KUKA KRL program: ap_0.src, ap_0.dat

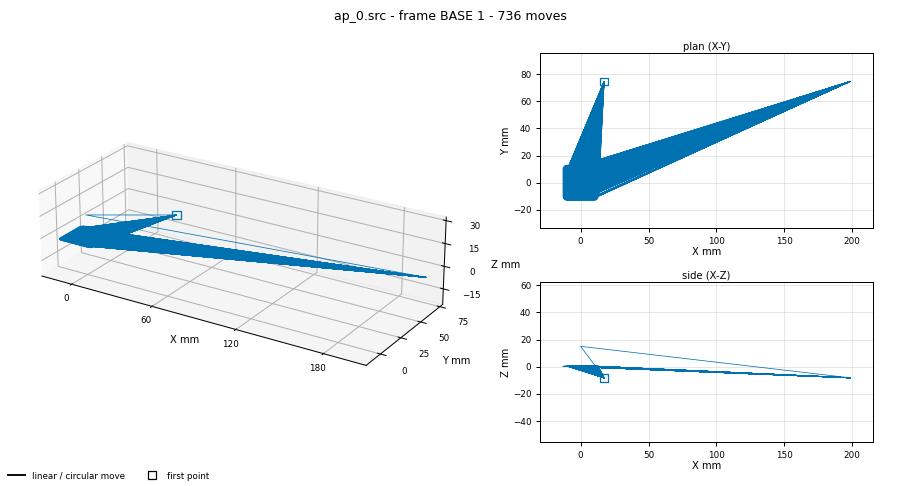
[picture p0: tool path of ap_0.src in frame BASE 1, 736 of 736 moves have a stored position in this frame; points joined in program order, loops and branches not executed]
--- ap_0.src ---
&ACCESS RVP
&REL 65
&PARAM DISKPATH = KRC:\R1\Program
DEF ap_0 ( )
   ;FOLD INI;%{PE}
     ;FOLD BASISTECH INI
       GLOBAL INTERRUPT DECL 3 WHEN $STOPMESS==TRUE DO IR_STOPM ( )
       INTERRUPT ON 3
       BAS (#INITMOV,0 )
     ;ENDFOLD (BASISTECH INI)
     ;FOLD USER INI
       ;Make your modifications here
     ;ENDFOLD (USER INI)
   ;ENDFOLD (INI)

   BAS (#VEL_PTP, 0020.0000)
   BAS (#ACC_PTP, 0020.0000)

   ;-----SET LIN AND ARC MOTION VARIABLES-----
   $VEL.ORI1 = 0350.0000
   $VEL.ORI2 = 0350.0000

   $ACC.CP = 0005.0000
   $ACC.ORI1 = 1000.0000
   $ACC.ORI2 = 1000.0000

   ;-----APPROXIMATION-----
   $APO.CVEL = 0100
   $APO.CPTP = 0100
   $APO.CDIS = 0006.0000
   $APO.CORI = 0090.0000

   BAS (#BASE, 1) ;Positioner
   BAS (#TOOL, 1) ;Vrashatel

   BAS(#VEL_PTP,15)                         ;;Set PTP Axis Velocity
   BAS(#ACC_PTP,50)                         ;;Set PTP Axis Acceleration
   PTP{A1 -92,A2 -133,A3 132,A4 7,A5 50,A6 -10}

;FOLD ARCON WDAT1 LIN P3 Vel=0.5 m/s CPDAT1 Tool[1]:cmttorch Base[1]:vrashatel ;%{PE}
  ;FOLD Parameters ;%{h}
    ;Params IlfProvider=kukaroboter.arctech.arconlin; Kuka.IsGlobalPoint=False; Kuka.PointName=P3; Kuka.BlendingEnabled=False; Kuka.MoveDataName=CPDAT1; Kuka.VelocityPath=0.5; Kuka.CurrentCDSetIndex=0; Kuka.MovementParameterFieldEnabled=True; ArcTech.WdatVarName=WDAT1; ArcTech.Basic=3.4.3.1264
  ;ENDFOLD
  $BWDSTART = FALSE
  LDAT_ACT = LCPDAT1
  FDAT_ACT = FP3
  BAS(#CP_PARAMS, 0.5)
  SET_CD_PARAMS (0)
  TRIGGER WHEN DISTANCE = 1 DELAY = ArcGetDelay(#PreDefinition, WDAT1) DO ArcMainNG(#PreDefinition, WDAT1, WP3) PRIO = -1
  TRIGGER WHEN PATH = ArcGetPath(#OnTheFlyArcOn, WDAT1) DELAY = ArcGetDelay(#GasPreflow, WDAT1) DO ArcMainNG(#GasPreflow, WDAT1, WP3) PRIO = -1
  TRIGGER WHEN PATH = ArcGetPath(#OnTheFlyArcOn, WDAT1) DELAY = 0 DO ArcMainNG(#ArcOnMoveStd, WDAT1, WP3) PRIO = -1
  ArcMainNG(#ArcOnBeforeMoveStd, WDAT1, WP3)
  LIN XP3
  ArcMainNG(#ArcOnAfterMoveStd, WDAT1, WP3)
;ENDFOLD
   $VEL.CP = 0.003
   LIN  {X 0.000, Y 0.000, Z 15.000, A 0.000, B 0.000, C 0.000} C_DIS

;FOLD ARCOFF WDAT2 LIN P4 CPDAT2 Tool[1]:cmttorch Base[1]:vrashatel ;%{PE}
  ;FOLD Parameters ;%{h}
    ;Params IlfProvider=kukaroboter.arctech.arcofflin; Kuka.IsGlobalPoint=False; Kuka.PointName=P4; Kuka.BlendingEnabled=False; Kuka.MoveDataName=CPDAT2; Kuka.VelocityPath=0.01; Kuka.CurrentCDSetIndex=0; Kuka.MovementParameterFieldEnabled=True; ArcTech.WdatVarName=WDAT2; ArcTech.Basic=3.4.3.1264
  ;ENDFOLD
  $BWDSTART = FALSE
  LDAT_ACT = LCPDAT2
  FDAT_ACT = FP4
  BAS(#CP_PARAMS, gArcBasVelDefinition)
  SET_CD_PARAMS (0)
  TRIGGER WHEN PATH = ArcGetPath(#ArcOffBefore, WDAT2) DELAY = 0 DO ArcMainNG(#ArcOffBeforeOffStd, WDAT2, WP4) PRIO = -1
  TRIGGER WHEN PATH = ArcGetPath(#OnTheFlyArcOff, WDAT2) DELAY = 0 DO ArcMainNG(#ArcOffMoveStd, WDAT2, WP4) PRIO = -1
  ArcMainNG(#ArcOffBeforeMoveStd, WDAT2, WP4)
  LIN XP4
  ArcMainNG(#ArcOffAfterMoveStd, WDAT2, WP4)
;ENDFOLD
   $VEL.CP = 0.030
   LIN  {X 13.000, Y -10.000, Z 0.300, A 0.000, B 0.000, C 0.000} C_DIS

;FOLD ARCON WDAT1 LIN P3 Vel=0.5 m/s CPDAT1 Tool[1]:cmttorch Base[1]:vrashatel ;%{PE}
  ;FOLD Parameters ;%{h}
    ;Params IlfProvider=kukaroboter.arctech.arconlin; Kuka.IsGlobalPoint=False; Kuka.PointName=P3; Kuka.BlendingEnabled=False; Kuka.MoveDataName=CPDAT1; Kuka.VelocityPath=0.5; Kuka.CurrentCDSetIndex=0; Kuka.MovementParameterFieldEnabled=True; ArcTech.WdatVarName=WDAT1; ArcTech.Basic=3.4.3.1264
  ;ENDFOLD
  $BWDSTART = FALSE
  LDAT_ACT = LCPDAT1
  FDAT_ACT = FP3
  BAS(#CP_PARAMS, 0.5)
  SET_CD_PARAMS (0)
  TRIGGER WHEN DISTANCE = 1 DELAY = ArcGetDelay(#PreDefinition, WDAT1) DO ArcMainNG(#PreDefinition, WDAT1, WP3) PRIO = -1
  TRIGGER WHEN PATH = ArcGetPath(#OnTheFlyArcOn, WDAT1) DELAY = ArcGetDelay(#GasPreflow, WDAT1) DO ArcMainNG(#GasPreflow, WDAT1, WP3) PRIO = -1
  TRIGGER WHEN PATH = ArcGetPath(#OnTheFlyArcOn, WDAT1) DELAY = 0 DO ArcMainNG(#ArcOnMoveStd, WDAT1, WP3) PRIO = -1
  ArcMainNG(#ArcOnBeforeMoveStd, WDAT1, WP3)
  LIN XP3
  ArcMainNG(#ArcOnAfterMoveStd, WDAT1, WP3)
;ENDFOLD
   $VEL.CP = 0.025
   LIN  {X 13.000, Y -10.000, Z 0.300, A 0.000, B 0.000, C 0.000} C_DIS
   $VEL.CP = 0.030
   LIN  {X 13.000, Y 10.000, Z 0.300, A 0.000, B 0.000, C 0.000} C_DIS
   $VEL.CP = 0.030
   LIN  {X 12.960, Y 10.488, Z 0.300, A 0.000, B 0.000, C 0.000} C_DIS
   $VEL.CP = 0.030
   LIN  {X 12.841, Y 10.963, Z 0.300, A 0.000, B 0.000, C 0.000} C_DIS
   $VEL.CP = 0.030
   LIN  {X 12.647, Y 11.412, Z 0.300, A 0.000, B 0.000, C 0.000} C_DIS
   $VEL.CP = 0.030
   LIN  {X 12.382, Y 11.824, Z 0.300, A 0.000, B 0.000, C 0.000} C_DIS
   $VEL.CP = 0.030
   LIN  {X 12.054, Y 12.187, Z 0.300, A 0.000, B 0.000, C 0.000} C_DIS
   $VEL.CP = 0.030
   LIN  {X 11.671, Y 12.492, Z 0.300, A 0.000, B 0.000, C 0.000} C_DIS
   $VEL.CP = 0.030
   LIN  {X 11.243, Y 12.730, Z 0.300, A 0.000, B 0.000, C 0.000} C_DIS
   $VEL.CP = 0.030
   LIN  {X 10.783, Y 12.896, Z 0.300, A 0.000, B 0.000, C 0.000} C_DIS
   $VEL.CP = 0.030
   LIN  {X 10.302, Y 12.985, Z 0.300, A 0.000, B 0.000, C 0.000} C_DIS
   $VEL.CP = 0.030
   LIN  {X 10.000, Y 13.000, Z 0.300, A 0.000, B 0.000, C 0.000} C_DIS
   $VEL.CP = 0.030
   LIN  {X -10.000, Y 13.000, Z 0.300, A 0.000, B 0.000, C 0.000} C_DIS
   $VEL.CP = 0.030
   LIN  {X -10.488, Y 12.960, Z 0.300, A 0.000, B 0.000, C 0.000} C_DIS
   $VEL.CP = 0.030
   LIN  {X -10.963, Y 12.841, Z 0.300, A 0.000, B 0.000, C 0.000} C_DIS
   $VEL.CP = 0.030
   LIN  {X -11.412, Y 12.647, Z 0.300, A 0.000, B 0.000, C 0.000} C_DIS
   $VEL.CP = 0.030
   LIN  {X -11.824, Y 12.382, Z 0.300, A 0.000, B 0.000, C 0.000} C_DIS
   $VEL.CP = 0.030
   LIN  {X -12.187, Y 12.054, Z 0.300, A 0.000, B 0.000, C 0.000} C_DIS
   $VEL.CP = 0.030
   LIN  {X -12.492, Y 11.671, Z 0.300, A 0.000, B 0.000, C 0.000} C_DIS
   $VEL.CP = 0.030
   LIN  {X -12.730, Y 11.243, Z 0.300, A 0.000, B 0.000, C 0.000} C_DIS
   $VEL.CP = 0.030
   LIN  {X -12.896, Y 10.783, Z 0.300, A 0.000, B 0.000, C 0.000} C_DIS
   $VEL.CP = 0.030
   LIN  {X -12.985, Y 10.302, Z 0.300, A 0.000, B 0.000, C 0.000} C_DIS
   $VEL.CP = 0.030
   LIN  {X -13.000, Y 10.000, Z 0.300, A 0.000, B 0.000, C 0.000} C_DIS
   $VEL.CP = 0.030
   LIN  {X -13.000, Y -10.000, Z 0.300, A 0.000, B 0.000, C 0.000} C_DIS
   $VEL.CP = 0.030
   LIN  {X -12.960, Y -10.488, Z 0.300, A 0.000, B 0.000, C 0.000} C_DIS
   $VEL.CP = 0.030
   LIN  {X -12.841, Y -10.963, Z 0.300, A 0.000, B 0.000, C 0.000} C_DIS
   $VEL.CP = 0.030
   LIN  {X -12.647, Y -11.412, Z 0.300, A 0.000, B 0.000, C 0.000} C_DIS
   $VEL.CP = 0.030
   LIN  {X -12.382, Y -11.824, Z 0.300, A 0.000, B 0.000, C 0.000} C_DIS
   $VEL.CP = 0.030
   LIN  {X -12.054, Y -12.187, Z 0.300, A 0.000, B 0.000, C 0.000} C_DIS
   $VEL.CP = 0.030
   LIN  {X -11.671, Y -12.492, Z 0.300, A 0.000, B 0.000, C 0.000} C_DIS
   $VEL.CP = 0.030
   LIN  {X -11.243, Y -12.730, Z 0.300, A 0.000, B 0.000, C 0.000} C_DIS
   $VEL.CP = 0.030
   LIN  {X -10.783, Y -12.896, Z 0.300, A 0.000, B 0.000, C 0.000} C_DIS
   $VEL.CP = 0.030
   LIN  {X -10.302, Y -12.985, Z 0.300, A 0.000, B 0.000, C 0.000} C_DIS
   $VEL.CP = 0.030
   LIN  {X -10.000, Y -13.000, Z 0.300, A 0.000, B 0.000, C 0.000} C_DIS
   $VEL.CP = 0.030
   LIN  {X 10.000, Y -13.000, Z 0.300, A 0.000, B 0.000, C 0.000} C_DIS
   $VEL.CP = 0.030
   LIN  {X 10.488, Y -12.960, Z 0.300, A 0.000, B 0.000, C 0.000} C_DIS
   $VEL.CP = 0.030
   LIN  {X 10.963, Y -12.841, Z 0.300, A 0.000, B 0.000, C 0.000} C_DIS
   $VEL.CP = 0.030
   LIN  {X 11.412, Y -12.647, Z 0.300, A 0.000, B 0.000, C 0.000} C_DIS
   $VEL.CP = 0.030
   LIN  {X 11.824, Y -12.382, Z 0.300, A 0.000, B 0.000, C 0.000} C_DIS
   $VEL.CP = 0.030
   LIN  {X 12.187, Y -12.054, Z 0.300, A 0.000, B 0.000, C 0.000} C_DIS
   $VEL.CP = 0.030
   LIN  {X 12.492, Y -11.671, Z 0.300, A 0.000, B 0.000, C 0.000} C_DIS
   $VEL.CP = 0.030
   LIN  {X 12.730, Y -11.243, Z 0.300, A 0.000, B 0.000, C 0.000} C_DIS
   $VEL.CP = 0.030
   LIN  {X 12.896, Y -10.783, Z 0.300, A 0.000, B 0.000, C 0.000} C_DIS
   $VEL.CP = 0.030
   LIN  {X 12.985, Y -10.302, Z 0.300, A 0.000, B 0.000, C 0.000} C_DIS
   $VEL.CP = 0.030
   LIN  {X 13.000, Y -10.000, Z 0.300, A 0.000, B 0.000, C 0.000} C_DIS

;FOLD ARCOFF WDAT2 LIN P4 CPDAT2 Tool[1]:cmttorch Base[1]:vrashatel ;%{PE}
  ;FOLD Parameters ;%{h}
    ;Params IlfProvider=kukaroboter.arctech.arcofflin; Kuka.IsGlobalPoint=False; Kuka.PointName=P4; Kuka.BlendingEnabled=False; Kuka.MoveDataName=CPDAT2; Kuka.VelocityPath=0.01; Kuka.CurrentCDSetIndex=0; Kuka.MovementParameterFieldEnabled=True; ArcTech.WdatVarName=WDAT2; ArcTech.Basic=3.4.3.1264
  ;ENDFOLD
  $BWDSTART = FALSE
  LDAT_ACT = LCPDAT2
  FDAT_ACT = FP4
  BAS(#CP_PARAMS, gArcBasVelDefinition)
  SET_CD_PARAMS (0)
  TRIGGER WHEN PATH = ArcGetPath(#ArcOffBefore, WDAT2) DELAY = 0 DO ArcMainNG(#ArcOffBeforeOffStd, WDAT2, WP4) PRIO = -1
  TRIGGER WHEN PATH = ArcGetPath(#OnTheFlyArcOff, WDAT2) DELAY = 0 DO ArcMainNG(#ArcOffMoveStd, WDAT2, WP4) PRIO = -1
  ArcMainNG(#ArcOffBeforeMoveStd, WDAT2, WP4)
  LIN XP4
  ArcMainNG(#ArcOffAfterMoveStd, WDAT2, WP4)
;ENDFOLD
   $VEL.CP = 0.030
   LIN  {X 12.600, Y -10.000, Z 0.300, A 0.000, B 0.000, C 0.000} C_DIS

;FOLD ARCON WDAT1 LIN P3 Vel=0.5 m/s CPDAT1 Tool[1]:cmttorch Base[1]:vrashatel ;%{PE}
  ;FOLD Parameters ;%{h}
    ;Params IlfProvider=kukaroboter.arctech.arconlin; Kuka.IsGlobalPoint=False; Kuka.PointName=P3; Kuka.BlendingEnabled=False; Kuka.MoveDataName=CPDAT1; Kuka.VelocityPath=0.5; Kuka.CurrentCDSetIndex=0; Kuka.MovementParameterFieldEnabled=True; ArcTech.WdatVarName=WDAT1; ArcTech.Basic=3.4.3.1264
  ;ENDFOLD
  $BWDSTART = FALSE
  LDAT_ACT = LCPDAT1
  FDAT_ACT = FP3
  BAS(#CP_PARAMS, 0.5)
  SET_CD_PARAMS (0)
  TRIGGER WHEN DISTANCE = 1 DELAY = ArcGetDelay(#PreDefinition, WDAT1) DO ArcMainNG(#PreDefinition, WDAT1, WP3) PRIO = -1
  TRIGGER WHEN PATH = ArcGetPath(#OnTheFlyArcOn, WDAT1) DELAY = ArcGetDelay(#GasPreflow, WDAT1) DO ArcMainNG(#GasPreflow, WDAT1, WP3) PRIO = -1
  TRIGGER WHEN PATH = ArcGetPath(#OnTheFlyArcOn, WDAT1) DELAY = 0 DO ArcMainNG(#ArcOnMoveStd, WDAT1, WP3) PRIO = -1
  ArcMainNG(#ArcOnBeforeMoveStd, WDAT1, WP3)
  LIN XP3
  ArcMainNG(#ArcOnAfterMoveStd, WDAT1, WP3)
;ENDFOLD
   $VEL.CP = 0.030
   LIN  {X 12.600, Y 10.000, Z 0.300, A 0.000, B 0.000, C 0.000} C_DIS
   $VEL.CP = 0.030
   LIN  {X 12.560, Y 10.454, Z 0.300, A 0.000, B 0.000, C 0.000} C_DIS
   $VEL.CP = 0.030
   LIN  {X 12.442, Y 10.894, Z 0.300, A 0.000, B 0.000, C 0.000} C_DIS
   $VEL.CP = 0.030
   LIN  {X 12.248, Y 11.306, Z 0.300, A 0.000, B 0.000, C 0.000} C_DIS
   $VEL.CP = 0.030
   LIN  {X 11.985, Y 11.679, Z 0.300, A 0.000, B 0.000, C 0.000} C_DIS
   $VEL.CP = 0.030
   LIN  {X 11.662, Y 12.000, Z 0.300, A 0.000, B 0.000, C 0.000} C_DIS
   $VEL.CP = 0.030
   LIN  {X 11.287, Y 12.259, Z 0.300, A 0.000, B 0.000, C 0.000} C_DIS
   $VEL.CP = 0.030
   LIN  {X 10.873, Y 12.449, Z 0.300, A 0.000, B 0.000, C 0.000} C_DIS
   $VEL.CP = 0.030
   LIN  {X 10.432, Y 12.564, Z 0.300, A 0.000, B 0.000, C 0.000} C_DIS
   $VEL.CP = 0.030
   LIN  {X 10.000, Y 12.600, Z 0.300, A 0.000, B 0.000, C 0.000} C_DIS
   $VEL.CP = 0.030
   LIN  {X -10.000, Y 12.600, Z 0.300, A 0.000, B 0.000, C 0.000} C_DIS
   $VEL.CP = 0.030
   LIN  {X -10.454, Y 12.560, Z 0.300, A 0.000, B 0.000, C 0.000} C_DIS
   $VEL.CP = 0.030
   LIN  {X -10.894, Y 12.442, Z 0.300, A 0.000, B 0.000, C 0.000} C_DIS
   $VEL.CP = 0.030
   LIN  {X -11.306, Y 12.248, Z 0.300, A 0.000, B 0.000, C 0.000} C_DIS
   $VEL.CP = 0.030
   LIN  {X -11.679, Y 11.985, Z 0.300, A 0.000, B 0.000, C 0.000} C_DIS
   $VEL.CP = 0.030
   LIN  {X -12.000, Y 11.662, Z 0.300, A 0.000, B 0.000, C 0.000} C_DIS
   $VEL.CP = 0.030
   LIN  {X -12.259, Y 11.287, Z 0.300, A 0.000, B 0.000, C 0.000} C_DIS
   $VEL.CP = 0.030
   LIN  {X -12.449, Y 10.873, Z 0.300, A 0.000, B 0.000, C 0.000} C_DIS
   $VEL.CP = 0.030
   LIN  {X -12.564, Y 10.432, Z 0.300, A 0.000, B 0.000, C 0.000} C_DIS
   $VEL.CP = 0.030
   LIN  {X -12.600, Y 10.000, Z 0.300, A 0.000, B 0.000, C 0.000} C_DIS
   $VEL.CP = 0.030
   LIN  {X -12.600, Y -10.000, Z 0.300, A 0.000, B 0.000, C 0.000} C_DIS
   $VEL.CP = 0.030
   LIN  {X -12.560, Y -10.454, Z 0.300, A 0.000, B 0.000, C 0.000} C_DIS
   $VEL.CP = 0.030
   LIN  {X -12.442, Y -10.894, Z 0.300, A 0.000, B 0.000, C 0.000} C_DIS
   $VEL.CP = 0.030
   LIN  {X -12.248, Y -11.306, Z 0.300, A 0.000, B 0.000, C 0.000} C_DIS
   $VEL.CP = 0.030
   LIN  {X -11.985, Y -11.679, Z 0.300, A 0.000, B 0.000, C 0.000} C_DIS
   $VEL.CP = 0.030
   LIN  {X -11.662, Y -12.000, Z 0.300, A 0.000, B 0.000, C 0.000} C_DIS
   $VEL.CP = 0.030
   LIN  {X -11.287, Y -12.259, Z 0.300, A 0.000, B 0.000, C 0.000} C_DIS
   $VEL.CP = 0.030
   LIN  {X -10.873, Y -12.449, Z 0.300, A 0.000, B 0.000, C 0.000} C_DIS
   $VEL.CP = 0.030
   LIN  {X -10.432, Y -12.564, Z 0.300, A 0.000, B 0.000, C 0.000} C_DIS
   $VEL.CP = 0.030
   LIN  {X -10.000, Y -12.600, Z 0.300, A 0.000, B 0.000, C 0.000} C_DIS
   $VEL.CP = 0.030
   LIN  {X 10.000, Y -12.600, Z 0.300, A 0.000, B 0.000, C 0.000} C_DIS
   $VEL.CP = 0.030
   LIN  {X 10.454, Y -12.560, Z 0.300, A 0.000, B 0.000, C 0.000} C_DIS
   $VEL.CP = 0.030
   LIN  {X 10.894, Y -12.442, Z 0.300, A 0.000, B 0.000, C 0.000} C_DIS
   $VEL.CP = 0.030
   LIN  {X 11.306, Y -12.248, Z 0.300, A 0.000, B 0.000, C 0.000} C_DIS
   $VEL.CP = 0.030
   LIN  {X 11.679, Y -11.985, Z 0.300, A 0.000, B 0.000, C 0.000} C_DIS
   $VEL.CP = 0.030
   LIN  {X 12.000, Y -11.662, Z 0.300, A 0.000, B 0.000, C 0.000} C_DIS
   $VEL.CP = 0.030
   LIN  {X 12.259, Y -11.287, Z 0.300, A 0.000, B 0.000, C 0.000} C_DIS
   $VEL.CP = 0.030
   LIN  {X 12.449, Y -10.873, Z 0.300, A 0.000, B 0.000, C 0.000} C_DIS
   $VEL.CP = 0.030
   LIN  {X 12.564, Y -10.432, Z 0.300, A 0.000, B 0.000, C 0.000} C_DIS
   $VEL.CP = 0.030
   LIN  {X 12.600, Y -10.000, Z 0.300, A 0.000, B 0.000, C 0.000} C_DIS

;FOLD ARCOFF WDAT2 LIN P4 CPDAT2 Tool[1]:cmttorch Base[1]:vrashatel ;%{PE}
  ;FOLD Parameters ;%{h}
    ;Params IlfProvider=kukaroboter.arctech.arcofflin; Kuka.IsGlobalPoint=False; Kuka.PointName=P4; Kuka.BlendingEnabled=False; Kuka.MoveDataName=CPDAT2; Kuka.VelocityPath=0.01; Kuka.CurrentCDSetIndex=0; Kuka.MovementParameterFieldEnabled=True; ArcTech.WdatVarName=WDAT2; ArcTech.Basic=3.4.3.1264
  ;ENDFOLD
  $BWDSTART = FALSE
  LDAT_ACT = LCPDAT2
  FDAT_ACT = FP4
  BAS(#CP_PARAMS, gArcBasVelDefinition)
  SET_CD_PARAMS (0)
  TRIGGER WHEN PATH = ArcGetPath(#ArcOffBefore, WDAT2) DELAY = 0 DO ArcMainNG(#ArcOffBeforeOffStd, WDAT2, WP4) PRIO = -1
  TRIGGER WHEN PATH = ArcGetPath(#OnTheFlyArcOff, WDAT2) DELAY = 0 DO ArcMainNG(#ArcOffMoveStd, WDAT2, WP4) PRIO = -1
  ArcMainNG(#ArcOffBeforeMoveStd, WDAT2, WP4)
  LIN XP4
  ArcMainNG(#ArcOffAfterMoveStd, WDAT2, WP4)
;ENDFOLD
   $VEL.CP = 0.030
   LIN  {X 12.200, Y -10.000, Z 0.300, A 0.000, B 0.000, C 0.000} C_DIS

;FOLD ARCON WDAT1 LIN P3 Vel=0.5 m/s CPDAT1 Tool[1]:cmttorch Base[1]:vrashatel ;%{PE}
  ;FOLD Parameters ;%{h}
    ;Params IlfProvider=kukaroboter.arctech.arconlin; Kuka.IsGlobalPoint=False; Kuka.PointName=P3; Kuka.BlendingEnabled=False; Kuka.MoveDataName=CPDAT1; Kuka.VelocityPath=0.5; Kuka.CurrentCDSetIndex=0; Kuka.MovementParameterFieldEnabled=True; ArcTech.WdatVarName=WDAT1; ArcTech.Basic=3.4.3.1264
  ;ENDFOLD
  $BWDSTART = FALSE
  LDAT_ACT = LCPDAT1
  FDAT_ACT = FP3
  BAS(#CP_PARAMS, 0.5)
  SET_CD_PARAMS (0)
  TRIGGER WHEN DISTANCE = 1 DELAY = ArcGetDelay(#PreDefinition, WDAT1) DO ArcMainNG(#PreDefinition, WDAT1, WP3) PRIO = -1
  TRIGGER WHEN PATH = ArcGetPath(#OnTheFlyArcOn, WDAT1) DELAY = ArcGetDelay(#GasPreflow, WDAT1) DO ArcMainNG(#GasPreflow, WDAT1, WP3) PRIO = -1
  TRIGGER WHEN PATH = ArcGetPath(#OnTheFlyArcOn, WDAT1) DELAY = 0 DO ArcMainNG(#ArcOnMoveStd, WDAT1, WP3) PRIO = -1
  ArcMainNG(#ArcOnBeforeMoveStd, WDAT1, WP3)
  LIN XP3
  ArcMainNG(#ArcOnAfterMoveStd, WDAT1, WP3)
;ENDFOLD
   $VEL.CP = 0.030
   LIN  {X 12.200, Y 10.000, Z 0.300, A 0.000, B 0.000, C 0.000} C_DIS
   $VEL.CP = 0.030
   LIN  {X 12.160, Y 10.417, Z 0.300, A 0.000, B 0.000, C 0.000} C_DIS
   $VEL.CP = 0.030
   LIN  {X 12.042, Y 10.819, Z 0.300, A 0.000, B 0.000, C 0.000} C_DIS
   $VEL.CP = 0.030
   LIN  {X 11.849, Y 11.191, Z 0.300, A 0.000, B 0.000, C 0.000} C_DIS
   $VEL.CP = 0.030
   LIN  {X 11.590, Y 11.520, Z 0.300, A 0.000, B 0.000, C 0.000} C_DIS
   $VEL.CP = 0.030
   LIN  {X 11.273, Y 11.794, Z 0.300, A 0.000, B 0.000, C 0.000} C_DIS
   $VEL.CP = 0.030
   LIN  {X 10.910, Y 12.003, Z 0.300, A 0.000, B 0.000, C 0.000} C_DIS
   $VEL.CP = 0.030
   LIN  {X 10.513, Y 12.139, Z 0.300, A 0.000, B 0.000, C 0.000} C_DIS
   $VEL.CP = 0.030
   LIN  {X 10.000, Y 12.200, Z 0.300, A 0.000, B 0.000, C 0.000} C_DIS
   $VEL.CP = 0.030
   LIN  {X -10.000, Y 12.200, Z 0.300, A 0.000, B 0.000, C 0.000} C_DIS
   $VEL.CP = 0.030
   LIN  {X -10.417, Y 12.160, Z 0.300, A 0.000, B 0.000, C 0.000} C_DIS
   $VEL.CP = 0.030
   LIN  {X -10.819, Y 12.042, Z 0.300, A 0.000, B 0.000, C 0.000} C_DIS
   $VEL.CP = 0.030
   LIN  {X -11.191, Y 11.849, Z 0.300, A 0.000, B 0.000, C 0.000} C_DIS
   $VEL.CP = 0.030
   LIN  {X -11.520, Y 11.590, Z 0.300, A 0.000, B 0.000, C 0.000} C_DIS
   $VEL.CP = 0.030
   LIN  {X -11.794, Y 11.273, Z 0.300, A 0.000, B 0.000, C 0.000} C_DIS
   $VEL.CP = 0.030
   LIN  {X -12.003, Y 10.910, Z 0.300, A 0.000, B 0.000, C 0.000} C_DIS
   $VEL.CP = 0.030
   LIN  {X -12.139, Y 10.513, Z 0.300, A 0.000, B 0.000, C 0.000} C_DIS
   $VEL.CP = 0.030
   LIN  {X -12.200, Y 10.000, Z 0.300, A 0.000, B 0.000, C 0.000} C_DIS
   $VEL.CP = 0.030
   LIN  {X -12.200, Y -10.000, Z 0.300, A 0.000, B 0.000, C 0.000} C_DIS
   $VEL.CP = 0.030
   LIN  {X -12.160, Y -10.417, Z 0.300, A 0.000, B 0.000, C 0.000} C_DIS
   $VEL.CP = 0.030
   LIN  {X -12.042, Y -10.819, Z 0.300, A 0.000, B 0.000, C 0.000} C_DIS
   $VEL.CP = 0.030
   LIN  {X -11.849, Y -11.191, Z 0.300, A 0.000, B 0.000, C 0.000} C_DIS
   $VEL.CP = 0.030
   LIN  {X -11.590, Y -11.520, Z 0.300, A 0.000, B 0.000, C 0.000} C_DIS
   $VEL.CP = 0.030
   LIN  {X -11.273, Y -11.794, Z 0.300, A 0.000, B 0.000, C 0.000} C_DIS
   $VEL.CP = 0.030
   LIN  {X -10.910, Y -12.003, Z 0.300, A 0.000, B 0.000, C 0.000} C_DIS
   $VEL.CP = 0.030
   LIN  {X -10.513, Y -12.139, Z 0.300, A 0.000, B 0.000, C 0.000} C_DIS
   $VEL.CP = 0.030
   LIN  {X -10.000, Y -12.200, Z 0.300, A 0.000, B 0.000, C 0.000} C_DIS
   $VEL.CP = 0.030
   LIN  {X 10.000, Y -12.200, Z 0.300, A 0.000, B 0.000, C 0.000} C_DIS
   $VEL.CP = 0.030
   LIN  {X 10.417, Y -12.160, Z 0.300, A 0.000, B 0.000, C 0.000} C_DIS
   $VEL.CP = 0.030
   LIN  {X 10.819, Y -12.042, Z 0.300, A 0.000, B 0.000, C 0.000} C_DIS
   $VEL.CP = 0.030
   LIN  {X 11.191, Y -11.849, Z 0.300, A 0.000, B 0.000, C 0.000} C_DIS
   $VEL.CP = 0.030
   LIN  {X 11.520, Y -11.590, Z 0.300, A 0.000, B 0.000, C 0.000} C_DIS
   $VEL.CP = 0.030
   LIN  {X 11.794, Y -11.273, Z 0.300, A 0.000, B 0.000, C 0.000} C_DIS
   $VEL.CP = 0.030
   LIN  {X 12.003, Y -10.910, Z 0.300, A 0.000, B 0.000, C 0.000} C_DIS
   $VEL.CP = 0.030
   LIN  {X 12.139, Y -10.513, Z 0.300, A 0.000, B 0.000, C 0.000} C_DIS
   $VEL.CP = 0.030
   LIN  {X 12.200, Y -10.000, Z 0.300, A 0.000, B 0.000, C 0.000} C_DIS

;FOLD ARCOFF WDAT2 LIN P4 CPDAT2 Tool[1]:cmttorch Base[1]:vrashatel ;%{PE}
  ;FOLD Parameters ;%{h}
    ;Params IlfProvider=kukaroboter.arctech.arcofflin; Kuka.IsGlobalPoint=False; Kuka.PointName=P4; Kuka.BlendingEnabled=False; Kuka.MoveDataName=CPDAT2; Kuka.VelocityPath=0.01; Kuka.CurrentCDSetIndex=0; Kuka.MovementParameterFieldEnabled=True; ArcTech.WdatVarName=WDAT2; ArcTech.Basic=3.4.3.1264
  ;ENDFOLD
  $BWDSTART = FALSE
  LDAT_ACT = LCPDAT2
  FDAT_ACT = FP4
  BAS(#CP_PARAMS, gArcBasVelDefinition)
  SET_CD_PARAMS (0)
  TRIGGER WHEN PATH = ArcGetPath(#ArcOffBefore, WDAT2) DELAY = 0 DO ArcMainNG(#ArcOffBeforeOffStd, WDAT2, WP4) PRIO = -1
  TRIGGER WHEN PATH = ArcGetPath(#OnTheFlyArcOff, WDAT2) DELAY = 0 DO ArcMainNG(#ArcOffMoveStd, WDAT2, WP4) PRIO = -1
  ArcMainNG(#ArcOffBeforeMoveStd, WDAT2, WP4)
  LIN XP4
  ArcMainNG(#ArcOffAfterMoveStd, WDAT2, WP4)
;ENDFOLD
   $VEL.CP = 0.030
   LIN  {X 11.800, Y -10.000, Z 0.300, A 0.000, B 0.000, C 0.000} C_DIS

;FOLD ARCON WDAT1 LIN P3 Vel=0.5 m/s CPDAT1 Tool[1]:cmttorch Base[1]:vrashatel ;%{PE}
  ;FOLD Parameters ;%{h}
    ;Params IlfProvider=kukaroboter.arctech.arconlin; Kuka.IsGlobalPoint=False; Kuka.PointName=P3; Kuka.BlendingEnabled=False; Kuka.MoveDataName=CPDAT1; Kuka.VelocityPath=0.5; Kuka.CurrentCDSetIndex=0; Kuka.MovementParameterFieldEnabled=True; ArcTech.WdatVarName=WDAT1; ArcTech.Basic=3.4.3.1264
  ;ENDFOLD
  $BWDSTART = FALSE
  LDAT_ACT = LCPDAT1
  FDAT_ACT = FP3
  BAS(#CP_PARAMS, 0.5)
  SET_CD_PARAMS (0)
  TRIGGER WHEN DISTANCE = 1 DELAY = ArcGetDelay(#PreDefinition, WDAT1) DO ArcMainNG(#PreDefinition, WDAT1, WP3) PRIO = -1
  TRIGGER WHEN PATH = ArcGetPath(#OnTheFlyArcOn, WDAT1) DELAY = ArcGetDelay(#GasPreflow, WDAT1) DO ArcMainNG(#GasPreflow, WDAT1, WP3) PRIO = -1
  TRIGGER WHEN PATH = ArcGetPath(#OnTheFlyArcOn, WDAT1) DELAY = 0 DO ArcMainNG(#ArcOnMoveStd, WDAT1, WP3) PRIO = -1
  ArcMainNG(#ArcOnBeforeMoveStd, WDAT1, WP3)
  LIN XP3
  ArcMainNG(#ArcOnAfterMoveStd, WDAT1, WP3)
;ENDFOLD
   $VEL.CP = 0.030
   LIN  {X 11.800, Y 10.000, Z 0.300, A 0.000, B 0.000, C 0.000} C_DIS
   $VEL.CP = 0.030
   LIN  {X 11.760, Y 10.377, Z 0.300, A 0.000, B 0.000, C 0.000} C_DIS
   $VEL.CP = 0.030
   LIN  {X 11.642, Y 10.737, Z 0.300, A 0.000, B 0.000, C 0.000} C_DIS
   $VEL.CP = 0.030
   LIN  {X 11.452, Y 11.064, Z 0.300, A 0.000, B 0.000, C 0.000} C_DIS
   $VEL.CP = 0.030
   LIN  {X 11.197, Y 11.345, Z 0.300, A 0.000, B 0.000, C 0.000} C_DIS
   $VEL.CP = 0.030
   LIN  {X 10.888, Y 11.565, Z 0.300, A 0.000, B 0.000, C 0.000} C_DIS
   $VEL.CP = 0.030
   LIN  {X 10.541, Y 11.717, Z 0.300, A 0.000, B 0.000, C 0.000} C_DIS
   $VEL.CP = 0.030
   LIN  {X 10.000, Y 11.800, Z 0.300, A 0.000, B 0.000, C 0.000} C_DIS
   $VEL.CP = 0.030
   LIN  {X -10.000, Y 11.800, Z 0.300, A 0.000, B 0.000, C 0.000} C_DIS
   $VEL.CP = 0.030
   LIN  {X -10.377, Y 11.760, Z 0.300, A 0.000, B 0.000, C 0.000} C_DIS
   $VEL.CP = 0.030
   LIN  {X -10.737, Y 11.642, Z 0.300, A 0.000, B 0.000, C 0.000} C_DIS
   $VEL.CP = 0.030
   LIN  {X -11.064, Y 11.452, Z 0.300, A 0.000, B 0.000, C 0.000} C_DIS
   $VEL.CP = 0.030
   LIN  {X -11.345, Y 11.197, Z 0.300, A 0.000, B 0.000, C 0.000} C_DIS
   $VEL.CP = 0.030
   LIN  {X -11.565, Y 10.888, Z 0.300, A 0.000, B 0.000, C 0.000} C_DIS
   $VEL.CP = 0.030
   LIN  {X -11.717, Y 10.541, Z 0.300, A 0.000, B 0.000, C 0.000} C_DIS
   $VEL.CP = 0.030
   LIN  {X -11.800, Y 10.000, Z 0.300, A 0.000, B 0.000, C 0.000} C_DIS
   $VEL.CP = 0.030
   LIN  {X -11.800, Y -10.000, Z 0.300, A 0.000, B 0.000, C 0.000} C_DIS
   $VEL.CP = 0.030
   LIN  {X -11.760, Y -10.377, Z 0.300, A 0.000, B 0.000, C 0.000} C_DIS
   $VEL.CP = 0.030
   LIN  {X -11.642, Y -10.737, Z 0.300, A 0.000, B 0.000, C 0.000} C_DIS
   $VEL.CP = 0.030
   LIN  {X -11.452, Y -11.064, Z 0.300, A 0.000, B 0.000, C 0.000} C_DIS
   $VEL.CP = 0.030
   LIN  {X -11.197, Y -11.345, Z 0.300, A 0.000, B 0.000, C 0.000} C_DIS
   $VEL.CP = 0.030
   LIN  {X -10.888, Y -11.565, Z 0.300, A 0.000, B 0.000, C 0.000} C_DIS
   $VEL.CP = 0.030
   LIN  {X -10.541, Y -11.717, Z 0.300, A 0.000, B 0.000, C 0.000} C_DIS
   $VEL.CP = 0.030
   LIN  {X -10.000, Y -11.800, Z 0.300, A 0.000, B 0.000, C 0.000} C_DIS
   $VEL.CP = 0.030
   LIN  {X 10.000, Y -11.800, Z 0.300, A 0.000, B 0.000, C 0.000} C_DIS
   $VEL.CP = 0.030
   LIN  {X 10.377, Y -11.760, Z 0.300, A 0.000, B 0.000, C 0.000} C_DIS
   $VEL.CP = 0.030
   LIN  {X 10.737, Y -11.642, Z 0.300, A 0.000, B 0.000, C 0.000} C_DIS
   $VEL.CP = 0.030
   LIN  {X 11.064, Y -11.452, Z 0.300, A 0.000, B 0.000, C 0.000} C_DIS
   $VEL.CP = 0.030
   LIN  {X 11.345, Y -11.197, Z 0.300, A 0.000, B 0.000, C 0.000} C_DIS
   $VEL.CP = 0.030
   LIN  {X 11.565, Y -10.888, Z 0.300, A 0.000, B 0.000, C 0.000} C_DIS
   $VEL.CP = 0.030
   LIN  {X 11.717, Y -10.541, Z 0.300, A 0.000, B 0.000, C 0.000} C_DIS
   $VEL.CP = 0.030
   LIN  {X 11.800, Y -10.000, Z 0.300, A 0.000, B 0.000, C 0.000} C_DIS

;FOLD ARCOFF WDAT2 LIN P4 CPDAT2 Tool[1]:cmttorch Base[1]:vrashatel ;%{PE}
  ;FOLD Parameters ;%{h}
    ;Params IlfProvider=kukaroboter.arctech.arcofflin; Kuka.IsGlobalPoint=False; Kuka.PointName=P4; Kuka.BlendingEnabled=False; Kuka.MoveDataName=CPDAT2; Kuka.VelocityPath=0.01; Kuka.CurrentCDSetIndex=0; Kuka.MovementParameterFieldEnabled=True; ArcTech.WdatVarName=WDAT2; ArcTech.Basic=3.4.3.1264
  ;ENDFOLD
  $BWDSTART = FALSE
  LDAT_ACT = LCPDAT2
  FDAT_ACT = FP4
  BAS(#CP_PARAMS, gArcBasVelDefinition)
  SET_CD_PARAMS (0)
  TRIGGER WHEN PATH = ArcGetPath(#ArcOffBefore, WDAT2) DELAY = 0 DO ArcMainNG(#ArcOffBeforeOffStd, WDAT2, WP4) PRIO = -1
  TRIGGER WHEN PATH = ArcGetPath(#OnTheFlyArcOff, WDAT2) DELAY = 0 DO ArcMainNG(#ArcOffMoveStd, WDAT2, WP4) PRIO = -1
  ArcMainNG(#ArcOffBeforeMoveStd, WDAT2, WP4)
  LIN XP4
  ArcMainNG(#ArcOffAfterMoveStd, WDAT2, WP4)
;ENDFOLD
   $VEL.CP = 0.030
   LIN  {X 11.400, Y -10.000, Z 0.300, A 0.000, B 0.000, C 0.000} C_DIS

;FOLD ARCON WDAT1 LIN P3 Vel=0.5 m/s CPDAT1 Tool[1]:cmttorch Base[1]:vrashatel ;%{PE}
  ;FOLD Parameters ;%{h}
    ;Params IlfProvider=kukaroboter.arctech.arconlin; Kuka.IsGlobalPoint=False; Kuka.PointName=P3; Kuka.BlendingEnabled=False; Kuka.MoveDataName=CPDAT1; Kuka.VelocityPath=0.5; Kuka.CurrentCDSetIndex=0; Kuka.MovementParameterFieldEnabled=True; ArcTech.WdatVarName=WDAT1; ArcTech.Basic=3.4.3.1264
  ;ENDFOLD
  $BWDSTART = FALSE
  LDAT_ACT = LCPDAT1
  FDAT_ACT = FP3
  BAS(#CP_PARAMS, 0.5)
  SET_CD_PARAMS (0)
  TRIGGER WHEN DISTANCE = 1 DELAY = ArcGetDelay(#PreDefinition, WDAT1) DO ArcMainNG(#PreDefinition, WDAT1, WP3) PRIO = -1
  TRIGGER WHEN PATH = ArcGetPath(#OnTheFlyArcOn, WDAT1) DELAY = ArcGetDelay(#GasPreflow, WDAT1) DO ArcMainNG(#GasPreflow, WDAT1, WP3) PRIO = -1
  TRIGGER WHEN PATH = ArcGetPath(#OnTheFlyArcOn, WDAT1) DELAY = 0 DO ArcMainNG(#ArcOnMoveStd, WDAT1, WP3) PRIO = -1
  ArcMainNG(#ArcOnBeforeMoveStd, WDAT1, WP3)
  LIN XP3
  ArcMainNG(#ArcOnAfterMoveStd, WDAT1, WP3)
;ENDFOLD
   $VEL.CP = 0.030
   LIN  {X 11.400, Y 10.000, Z 0.300, A 0.000, B 0.000, C 0.000} C_DIS
   $VEL.CP = 0.030
   LIN  {X 11.360, Y 10.332, Z 0.300, A 0.000, B 0.000, C 0.000} C_DIS
   $VEL.CP = 0.030
   LIN  {X 11.243, Y 10.644, Z 0.300, A 0.000, B 0.000, C 0.000} C_DIS
   $VEL.CP = 0.030
   LIN  {X 11.055, Y 10.921, Z 0.300, A 0.000, B 0.000, C 0.000} C_DIS
   $VEL.CP = 0.030
   LIN  {X 10.807, Y 11.144, Z 0.300, A 0.000, B 0.000, C 0.000} C_DIS
   $VEL.CP = 0.030
   LIN  {X 10.513, Y 11.303, Z 0.300, A 0.000, B 0.000, C 0.000} C_DIS
   $VEL.CP = 0.030
   LIN  {X 10.189, Y 11.387, Z 0.300, A 0.000, B 0.000, C 0.000} C_DIS
   $VEL.CP = 0.030
   LIN  {X 10.000, Y 11.400, Z 0.300, A 0.000, B 0.000, C 0.000} C_DIS
   $VEL.CP = 0.030
   LIN  {X -10.000, Y 11.400, Z 0.300, A 0.000, B 0.000, C 0.000} C_DIS
   $VEL.CP = 0.030
   LIN  {X -10.332, Y 11.360, Z 0.300, A 0.000, B 0.000, C 0.000} C_DIS
   $VEL.CP = 0.030
   LIN  {X -10.644, Y 11.243, Z 0.300, A 0.000, B 0.000, C 0.000} C_DIS
   $VEL.CP = 0.030
   LIN  {X -10.921, Y 11.055, Z 0.300, A 0.000, B 0.000, C 0.000} C_DIS
   $VEL.CP = 0.030
   LIN  {X -11.144, Y 10.807, Z 0.300, A 0.000, B 0.000, C 0.000} C_DIS
   $VEL.CP = 0.030
   LIN  {X -11.303, Y 10.513, Z 0.300, A 0.000, B 0.000, C 0.000} C_DIS
   $VEL.CP = 0.030
   LIN  {X -11.387, Y 10.189, Z 0.300, A 0.000, B 0.000, C 0.000} C_DIS
   $VEL.CP = 0.030
   LIN  {X -11.400, Y 10.000, Z 0.300, A 0.000, B 0.000, C 0.000} C_DIS
   $VEL.CP = 0.030
   LIN  {X -11.400, Y -10.000, Z 0.300, A 0.000, B 0.000, C 0.000} C_DIS
   $VEL.CP = 0.030
   LIN  {X -11.360, Y -10.332, Z 0.300, A 0.000, B 0.000, C 0.000} C_DIS
   $VEL.CP = 0.030
   LIN  {X -11.243, Y -10.644, Z 0.300, A 0.000, B 0.000, C 0.000} C_DIS
   $VEL.CP = 0.030
   LIN  {X -11.055, Y -10.921, Z 0.300, A 0.000, B 0.000, C 0.000} C_DIS
   $VEL.CP = 0.030
   LIN  {X -10.807, Y -11.144, Z 0.300, A 0.000, B 0.000, C 0.000} C_DIS
   $VEL.CP = 0.030
   LIN  {X -10.513, Y -11.303, Z 0.300, A 0.000, B 0.000, C 0.000} C_DIS
   $VEL.CP = 0.030
   LIN  {X -10.189, Y -11.387, Z 0.300, A 0.000, B 0.000, C 0.000} C_DIS
   $VEL.CP = 0.030
   LIN  {X -10.000, Y -11.400, Z 0.300, A 0.000, B 0.000, C 0.000} C_DIS
   $VEL.CP = 0.030
   LIN  {X 10.000, Y -11.400, Z 0.300, A 0.000, B 0.000, C 0.000} C_DIS
   $VEL.CP = 0.030
   LIN  {X 10.332, Y -11.360, Z 0.300, A 0.000, B 0.000, C 0.000} C_DIS
   $VEL.CP = 0.030
   LIN  {X 10.644, Y -11.243, Z 0.300, A 0.000, B 0.000, C 0.000} C_DIS
   $VEL.CP = 0.030
   LIN  {X 10.921, Y -11.055, Z 0.300, A 0.000, B 0.000, C 0.000} C_DIS
   $VEL.CP = 0.030
   LIN  {X 11.144, Y -10.807, Z 0.300, A 0.000, B 0.000, C 0.000} C_DIS
   $VEL.CP = 0.030
   LIN  {X 11.303, Y -10.513, Z 0.300, A 0.000, B 0.000, C 0.000} C_DIS
   $VEL.CP = 0.030
   LIN  {X 11.387, Y -10.189, Z 0.300, A 0.000, B 0.000, C 0.000} C_DIS
   $VEL.CP = 0.030
   LIN  {X 11.400, Y -10.000, Z 0.300, A 0.000, B 0.000, C 0.000} C_DIS

;FOLD ARCOFF WDAT2 LIN P4 CPDAT2 Tool[1]:cmttorch Base[1]:vrashatel ;%{PE}
  ;FOLD Parameters ;%{h}
    ;Params IlfProvider=kukaroboter.arctech.arcofflin; Kuka.IsGlobalPoint=False; Kuka.PointName=P4; Kuka.BlendingEnabled=False; Kuka.MoveDataName=CPDAT2; Kuka.VelocityPath=0.01; Kuka.CurrentCDSetIndex=0; Kuka.MovementParameterFieldEnabled=True; ArcTech.WdatVarName=WDAT2; ArcTech.Basic=3.4.3.1264
  ;ENDFOLD
  $BWDSTART = FALSE
  LDAT_ACT = LCPDAT2
  FDAT_ACT = FP4
  BAS(#CP_PARAMS, gArcBasVelDefinition)
  SET_CD_PARAMS (0)
  TRIGGER WHEN PATH = ArcGetPath(#ArcOffBefore, WDAT2) DELAY = 0 DO ArcMainNG(#ArcOffBeforeOffStd, WDAT2, WP4) PRIO = -1
  TRIGGER WHEN PATH = ArcGetPath(#OnTheFlyArcOff, WDAT2) DELAY = 0 DO ArcMainNG(#ArcOffMoveStd, WDAT2, WP4) PRIO = -1
  ArcMainNG(#ArcOffBeforeMoveStd, WDAT2, WP4)
  LIN XP4
  ArcMainNG(#ArcOffAfterMoveStd, WDAT2, WP4)
;ENDFOLD
   $VEL.CP = 0.030
   LIN  {X 11.000, Y -10.000, Z 0.300, A 0.000, B 0.000, C 0.000} C_DIS

;FOLD ARCON WDAT1 LIN P3 Vel=0.5 m/s CPDAT1 Tool[1]:cmttorch Base[1]:vrashatel ;%{PE}
  ;FOLD Parameters ;%{h}
    ;Params IlfProvider=kukaroboter.arctech.arconlin; Kuka.IsGlobalPoint=False; Kuka.PointName=P3; Kuka.BlendingEnabled=False; Kuka.MoveDataName=CPDAT1; Kuka.VelocityPath=0.5; Kuka.CurrentCDSetIndex=0; Kuka.MovementParameterFieldEnabled=True; ArcTech.WdatVarName=WDAT1; ArcTech.Basic=3.4.3.1264
  ;ENDFOLD
  $BWDSTART = FALSE
  LDAT_ACT = LCPDAT1
  FDAT_ACT = FP3
  BAS(#CP_PARAMS, 0.5)
  SET_CD_PARAMS (0)
  TRIGGER WHEN DISTANCE = 1 DELAY = ArcGetDelay(#PreDefinition, WDAT1) DO ArcMainNG(#PreDefinition, WDAT1, WP3) PRIO = -1
  TRIGGER WHEN PATH = ArcGetPath(#OnTheFlyArcOn, WDAT1) DELAY = ArcGetDelay(#GasPreflow, WDAT1) DO ArcMainNG(#GasPreflow, WDAT1, WP3) PRIO = -1
  TRIGGER WHEN PATH = ArcGetPath(#OnTheFlyArcOn, WDAT1) DELAY = 0 DO ArcMainNG(#ArcOnMoveStd, WDAT1, WP3) PRIO = -1
  ArcMainNG(#ArcOnBeforeMoveStd, WDAT1, WP3)
  LIN XP3
  ArcMainNG(#ArcOnAfterMoveStd, WDAT1, WP3)
;ENDFOLD
   $VEL.CP = 0.030
   LIN  {X 11.000, Y 10.000, Z 0.300, A 0.000, B 0.000, C 0.000} C_DIS
   $VEL.CP = 0.030
   LIN  {X 10.960, Y 10.279, Z 0.300, A 0.000, B 0.000, C 0.000} C_DIS
   $VEL.CP = 0.030
   LIN  {X 10.844, Y 10.536, Z 0.300, A 0.000, B 0.000, C 0.000} C_DIS
   $VEL.CP = 0.030
   LIN  {X 10.661, Y 10.751, Z 0.300, A 0.000, B 0.000, C 0.000} C_DIS
   $VEL.CP = 0.030
   LIN  {X 10.425, Y 10.905, Z 0.300, A 0.000, B 0.000, C 0.000} C_DIS
   $VEL.CP = 0.030
   LIN  {X 10.155, Y 10.988, Z 0.300, A 0.000, B 0.000, C 0.000} C_DIS
   $VEL.CP = 0.030
   LIN  {X 10.000, Y 11.000, Z 0.300, A 0.000, B 0.000, C 0.000} C_DIS
   $VEL.CP = 0.030
   LIN  {X -10.000, Y 11.000, Z 0.300, A 0.000, B 0.000, C 0.000} C_DIS
   $VEL.CP = 0.030
   LIN  {X -10.279, Y 10.960, Z 0.300, A 0.000, B 0.000, C 0.000} C_DIS
   $VEL.CP = 0.030
   LIN  {X -10.536, Y 10.844, Z 0.300, A 0.000, B 0.000, C 0.000} C_DIS
   $VEL.CP = 0.030
   LIN  {X -10.751, Y 10.661, Z 0.300, A 0.000, B 0.000, C 0.000} C_DIS
   $VEL.CP = 0.030
   LIN  {X -10.905, Y 10.425, Z 0.300, A 0.000, B 0.000, C 0.000} C_DIS
   $VEL.CP = 0.030
   LIN  {X -10.988, Y 10.155, Z 0.300, A 0.000, B 0.000, C 0.000} C_DIS
   $VEL.CP = 0.030
   LIN  {X -11.000, Y 10.000, Z 0.300, A 0.000, B 0.000, C 0.000} C_DIS
   $VEL.CP = 0.030
   LIN  {X -11.000, Y -10.000, Z 0.300, A 0.000, B 0.000, C 0.000} C_DIS
   $VEL.CP = 0.030
   LIN  {X -10.960, Y -10.279, Z 0.300, A 0.000, B 0.000, C 0.000} C_DIS
   $VEL.CP = 0.030
   LIN  {X -10.844, Y -10.536, Z 0.300, A 0.000, B 0.000, C 0.000} C_DIS
   $VEL.CP = 0.030
   LIN  {X -10.661, Y -10.751, Z 0.300, A 0.000, B 0.000, C 0.000} C_DIS
   $VEL.CP = 0.030
   LIN  {X -10.425, Y -10.905, Z 0.300, A 0.000, B 0.000, C 0.000} C_DIS
   $VEL.CP = 0.030
   LIN  {X -10.155, Y -10.988, Z 0.300, A 0.000, B 0.000, C 0.000} C_DIS
   $VEL.CP = 0.030
   LIN  {X -10.000, Y -11.000, Z 0.300, A 0.000, B 0.000, C 0.000} C_DIS
   $VEL.CP = 0.030
   LIN  {X 10.000, Y -11.000, Z 0.300, A 0.000, B 0.000, C 0.000} C_DIS
   $VEL.CP = 0.030
   LIN  {X 10.279, Y -10.960, Z 0.300, A 0.000, B 0.000, C 0.000} C_DIS
   $VEL.CP = 0.030
   LIN  {X 10.536, Y -10.844, Z 0.300, A 0.000, B 0.000, C 0.000} C_DIS
   $VEL.CP = 0.030
   LIN  {X 10.751, Y -10.661, Z 0.300, A 0.000, B 0.000, C 0.000} C_DIS
   $VEL.CP = 0.030
   LIN  {X 10.905, Y -10.425, Z 0.300, A 0.000, B 0.000, C 0.000} C_DIS
   $VEL.CP = 0.030
   LIN  {X 10.988, Y -10.155, Z 0.300, A 0.000, B 0.000, C 0.000} C_DIS
   $VEL.CP = 0.030
   LIN  {X 11.000, Y -10.000, Z 0.300, A 0.000, B 0.000, C 0.000} C_DIS

;FOLD ARCOFF WDAT2 LIN P4 CPDAT2 Tool[1]:cmttorch Base[1]:vrashatel ;%{PE}
  ;FOLD Parameters ;%{h}
    ;Params IlfProvider=kukaroboter.arctech.arcofflin; Kuka.IsGlobalPoint=False; Kuka.PointName=P4; Kuka.BlendingEnabled=False; Kuka.MoveDataName=CPDAT2; Kuka.VelocityPath=0.01; Kuka.CurrentCDSetIndex=0; Kuka.MovementParameterFieldEnabled=True; ArcTech.WdatVarName=WDAT2; ArcTech.Basic=3.4.3.1264
  ;ENDFOLD
  $BWDSTART = FALSE
  LDAT_ACT = LCPDAT2
  FDAT_ACT = FP4
  BAS(#CP_PARAMS, gArcBasVelDefinition)
  SET_CD_PARAMS (0)
  TRIGGER WHEN PATH = ArcGetPath(#ArcOffBefore, WDAT2) DELAY = 0 DO ArcMainNG(#ArcOffBeforeOffStd, WDAT2, WP4) PRIO = -1
  TRIGGER WHEN PATH = ArcGetPath(#OnTheFlyArcOff, WDAT2) DELAY = 0 DO ArcMainNG(#ArcOffMoveStd, WDAT2, WP4) PRIO = -1
  ArcMainNG(#ArcOffBeforeMoveStd, WDAT2, WP4)
  LIN XP4
  ArcMainNG(#ArcOffAfterMoveStd, WDAT2, WP4)
;ENDFOLD
   $VEL.CP = 0.030
   LIN  {X 10.600, Y -10.000, Z 0.300, A 0.000, B 0.000, C 0.000} C_DIS

;FOLD ARCON WDAT1 LIN P3 Vel=0.5 m/s CPDAT1 Tool[1]:cmttorch Base[1]:vrashatel ;%{PE}
  ;FOLD Parameters ;%{h}
    ;Params IlfProvider=kukaroboter.arctech.arconlin; Kuka.IsGlobalPoint=False; Kuka.PointName=P3; Kuka.BlendingEnabled=False; Kuka.MoveDataName=CPDAT1; Kuka.VelocityPath=0.5; Kuka.CurrentCDSetIndex=0; Kuka.MovementParameterFieldEnabled=True; ArcTech.WdatVarName=WDAT1; ArcTech.Basic=3.4.3.1264
  ;ENDFOLD
  $BWDSTART = FALSE
  LDAT_ACT = LCPDAT1
  FDAT_ACT = FP3
  BAS(#CP_PARAMS, 0.5)
  SET_CD_PARAMS (0)
  TRIGGER WHEN DISTANCE = 1 DELAY = ArcGetDelay(#PreDefinition, WDAT1) DO ArcMainNG(#PreDefinition, WDAT1, WP3) PRIO = -1
  TRIGGER WHEN PATH = ArcGetPath(#OnTheFlyArcOn, WDAT1) DELAY = ArcGetDelay(#GasPreflow, WDAT1) DO ArcMainNG(#GasPreflow, WDAT1, WP3) PRIO = -1
  TRIGGER WHEN PATH = ArcGetPath(#OnTheFlyArcOn, WDAT1) DELAY = 0 DO ArcMainNG(#ArcOnMoveStd, WDAT1, WP3) PRIO = -1
  ArcMainNG(#ArcOnBeforeMoveStd, WDAT1, WP3)
  LIN XP3
  ArcMainNG(#ArcOnAfterMoveStd, WDAT1, WP3)
;ENDFOLD
   $VEL.CP = 0.030
   LIN  {X 10.600, Y 10.000, Z 0.300, A 0.000, B 0.000, C 0.000} C_DIS
   $VEL.CP = 0.030
   LIN  {X 10.560, Y 10.215, Z 0.300, A 0.000, B 0.000, C 0.000} C_DIS
   $VEL.CP = 0.030
   LIN  {X 10.447, Y 10.401, Z 0.300, A 0.000, B 0.000, C 0.000} C_DIS
   $VEL.CP = 0.030
   LIN  {X 10.274, Y 10.534, Z 0.300, A 0.000, B 0.000, C 0.000} C_DIS
   $VEL.CP = 0.030
   LIN  {X 10.000, Y 10.600, Z 0.300, A 0.000, B 0.000, C 0.000} C_DIS
   $VEL.CP = 0.030
   LIN  {X -10.000, Y 10.600, Z 0.300, A 0.000, B 0.000, C 0.000} C_DIS
   $VEL.CP = 0.030
   LIN  {X -10.215, Y 10.560, Z 0.300, A 0.000, B 0.000, C 0.000} C_DIS
   $VEL.CP = 0.030
   LIN  {X -10.401, Y 10.447, Z 0.300, A 0.000, B 0.000, C 0.000} C_DIS
   $VEL.CP = 0.030
   LIN  {X -10.534, Y 10.274, Z 0.300, A 0.000, B 0.000, C 0.000} C_DIS
   $VEL.CP = 0.030
   LIN  {X -10.600, Y 10.000, Z 0.300, A 0.000, B 0.000, C 0.000} C_DIS
   $VEL.CP = 0.030
   LIN  {X -10.600, Y -10.000, Z 0.300, A 0.000, B 0.000, C 0.000} C_DIS
   $VEL.CP = 0.030
   LIN  {X -10.560, Y -10.215, Z 0.300, A 0.000, B 0.000, C 0.000} C_DIS
   $VEL.CP = 0.030
   LIN  {X -10.447, Y -10.401, Z 0.300, A 0.000, B 0.000, C 0.000} C_DIS
   $VEL.CP = 0.030
   LIN  {X -10.274, Y -10.534, Z 0.300, A 0.000, B 0.000, C 0.000} C_DIS
   $VEL.CP = 0.030
   LIN  {X -10.000, Y -10.600, Z 0.300, A 0.000, B 0.000, C 0.000} C_DIS
   $VEL.CP = 0.030
   LIN  {X 10.000, Y -10.600, Z 0.300, A 0.000, B 0.000, C 0.000} C_DIS
   $VEL.CP = 0.030
   LIN  {X 10.215, Y -10.560, Z 0.300, A 0.000, B 0.000, C 0.000} C_DIS
   $VEL.CP = 0.030
   LIN  {X 10.401, Y -10.447, Z 0.300, A 0.000, B 0.000, C 0.000} C_DIS
   $VEL.CP = 0.030
   LIN  {X 10.534, Y -10.274, Z 0.300, A 0.000, B 0.000, C 0.000} C_DIS
   $VEL.CP = 0.030
   LIN  {X 10.600, Y -10.000, Z 0.300, A 0.000, B 0.000, C 0.000} C_DIS

;FOLD ARCOFF WDAT2 LIN P4 CPDAT2 Tool[1]:cmttorch Base[1]:vrashatel ;%{PE}
  ;FOLD Parameters ;%{h}
    ;Params IlfProvider=kukaroboter.arctech.arcofflin; Kuka.IsGlobalPoint=False; Kuka.PointName=P4; Kuka.BlendingEnabled=False; Kuka.MoveDataName=CPDAT2; Kuka.VelocityPath=0.01; Kuka.CurrentCDSetIndex=0; Kuka.MovementParameterFieldEnabled=True; ArcTech.WdatVarName=WDAT2; ArcTech.Basic=3.4.3.1264
  ;ENDFOLD
  $BWDSTART = FALSE
  LDAT_ACT = LCPDAT2
  FDAT_ACT = FP4
  BAS(#CP_PARAMS, gArcBasVelDefinition)
  SET_CD_PARAMS (0)
  TRIGGER WHEN PATH = ArcGetPath(#ArcOffBefore, WDAT2) DELAY = 0 DO ArcMainNG(#ArcOffBeforeOffStd, WDAT2, WP4) PRIO = -1
  TRIGGER WHEN PATH = ArcGetPath(#OnTheFlyArcOff, WDAT2) DELAY = 0 DO ArcMainNG(#ArcOffMoveStd, WDAT2, WP4) PRIO = -1
  ArcMainNG(#ArcOffBeforeMoveStd, WDAT2, WP4)
  LIN XP4
  ArcMainNG(#ArcOffAfterMoveStd, WDAT2, WP4)
;ENDFOLD
   $VEL.CP = 0.030
   LIN  {X 10.200, Y -10.000, Z 0.300, A 0.000, B 0.000, C 0.000} C_DIS

;FOLD ARCON WDAT1 LIN P3 Vel=0.5 m/s CPDAT1 Tool[1]:cmttorch Base[1]:vrashatel ;%{PE}
  ;FOLD Parameters ;%{h}
    ;Params IlfProvider=kukaroboter.arctech.arconlin; Kuka.IsGlobalPoint=False; Kuka.PointName=P3; Kuka.BlendingEnabled=False; Kuka.MoveDataName=CPDAT1; Kuka.VelocityPath=0.5; Kuka.CurrentCDSetIndex=0; Kuka.MovementParameterFieldEnabled=True; ArcTech.WdatVarName=WDAT1; ArcTech.Basic=3.4.3.1264
  ;ENDFOLD
  $BWDSTART = FALSE
  LDAT_ACT = LCPDAT1
  FDAT_ACT = FP3
  BAS(#CP_PARAMS, 0.5)
  SET_CD_PARAMS (0)
  TRIGGER WHEN DISTANCE = 1 DELAY = ArcGetDelay(#PreDefinition, WDAT1) DO ArcMainNG(#PreDefinition, WDAT1, WP3) PRIO = -1
  TRIGGER WHEN PATH = ArcGetPath(#OnTheFlyArcOn, WDAT1) DELAY = ArcGetDelay(#GasPreflow, WDAT1) DO ArcMainNG(#GasPreflow, WDAT1, WP3) PRIO = -1
  TRIGGER WHEN PATH = ArcGetPath(#OnTheFlyArcOn, WDAT1) DELAY = 0 DO ArcMainNG(#ArcOnMoveStd, WDAT1, WP3) PRIO = -1
  ArcMainNG(#ArcOnBeforeMoveStd, WDAT1, WP3)
  LIN XP3
  ArcMainNG(#ArcOnAfterMoveStd, WDAT1, WP3)
;ENDFOLD
   $VEL.CP = 0.030
   LIN  {X 10.200, Y 10.000, Z 0.300, A 0.000, B 0.000, C 0.000} C_DIS
   $VEL.CP = 0.030
   LIN  {X 10.161, Y 10.119, Z 0.300, A 0.000, B 0.000, C 0.000} C_DIS
   $VEL.CP = 0.030
   LIN  {X 10.000, Y 10.200, Z 0.300, A 0.000, B 0.000, C 0.000} C_DIS
   $VEL.CP = 0.030
   LIN  {X -10.000, Y 10.200, Z 0.300, A 0.000, B 0.000, C 0.000} C_DIS
   $VEL.CP = 0.030
   LIN  {X -10.119, Y 10.161, Z 0.300, A 0.000, B 0.000, C 0.000} C_DIS
   $VEL.CP = 0.030
   LIN  {X -10.200, Y 10.000, Z 0.300, A 0.000, B 0.000, C 0.000} C_DIS
   $VEL.CP = 0.030
   LIN  {X -10.200, Y -10.000, Z 0.300, A 0.000, B 0.000, C 0.000} C_DIS
   $VEL.CP = 0.030
   LIN  {X -10.161, Y -10.119, Z 0.300, A 0.000, B 0.000, C 0.000} C_DIS
   $VEL.CP = 0.030
   LIN  {X -10.000, Y -10.200, Z 0.300, A 0.000, B 0.000, C 0.000} C_DIS
   $VEL.CP = 0.030
   LIN  {X 10.000, Y -10.200, Z 0.300, A 0.000, B 0.000, C 0.000} C_DIS
   $VEL.CP = 0.030
   LIN  {X 10.119, Y -10.161, Z 0.300, A 0.000, B 0.000, C 0.000} C_DIS
   $VEL.CP = 0.030
   LIN  {X 10.200, Y -10.000, Z 0.300, A 0.000, B 0.000, C 0.000} C_DIS

;FOLD ARCOFF WDAT2 LIN P4 CPDAT2 Tool[1]:cmttorch Base[1]:vrashatel ;%{PE}
  ;FOLD Parameters ;%{h}
    ;Params IlfProvider=kukaroboter.arctech.arcofflin; Kuka.IsGlobalPoint=False; Kuka.PointName=P4; Kuka.BlendingEnabled=False; Kuka.MoveDataName=CPDAT2; Kuka.VelocityPath=0.01; Kuka.CurrentCDSetIndex=0; Kuka.MovementParameterFieldEnabled=True; ArcTech.WdatVarName=WDAT2; ArcTech.Basic=3.4.3.1264
  ;ENDFOLD
  $BWDSTART = FALSE
  LDAT_ACT = LCPDAT2
  FDAT_ACT = FP4
  BAS(#CP_PARAMS, gArcBasVelDefinition)
  SET_CD_PARAMS (0)
  TRIGGER WHEN PATH = ArcGetPath(#ArcOffBefore, WDAT2) DELAY = 0 DO ArcMainNG(#ArcOffBeforeOffStd, WDAT2, WP4) PRIO = -1
  TRIGGER WHEN PATH = ArcGetPath(#OnTheFlyArcOff, WDAT2) DELAY = 0 DO ArcMainNG(#ArcOffMoveStd, WDAT2, WP4) PRIO = -1
  ArcMainNG(#ArcOffBeforeMoveStd, WDAT2, WP4)
  LIN XP4
  ArcMainNG(#ArcOffAfterMoveStd, WDAT2, WP4)
;ENDFOLD
   $VEL.CP = 0.030
   LIN  {X 9.190, Y -9.190, Z 0.300, A 0.000, B 0.000, C 0.000} C_DIS
   $VEL.CP = 0.030
   LIN  {X -9.500, Y 9.530, Z 0.300, A 0.000, B 0.000, C 0.000} C_DIS
   $VEL.CP = 0.030
   LIN  {X -9.800, Y 9.800, Z 0.300, A 0.000, B 0.000, C 0.000} C_DIS

;FOLD ARCON WDAT1 LIN P3 Vel=0.5 m/s CPDAT1 Tool[1]:cmttorch Base[1]:vrashatel ;%{PE}
  ;FOLD Parameters ;%{h}
    ;Params IlfProvider=kukaroboter.arctech.arconlin; Kuka.IsGlobalPoint=False; Kuka.PointName=P3; Kuka.BlendingEnabled=False; Kuka.MoveDataName=CPDAT1; Kuka.VelocityPath=0.5; Kuka.CurrentCDSetIndex=0; Kuka.MovementParameterFieldEnabled=True; ArcTech.WdatVarName=WDAT1; ArcTech.Basic=3.4.3.1264
  ;ENDFOLD
  $BWDSTART = FALSE
  LDAT_ACT = LCPDAT1
  FDAT_ACT = FP3
  BAS(#CP_PARAMS, 0.5)
  SET_CD_PARAMS (0)
  TRIGGER WHEN DISTANCE = 1 DELAY = ArcGetDelay(#PreDefinition, WDAT1) DO ArcMainNG(#PreDefinition, WDAT1, WP3) PRIO = -1
  TRIGGER WHEN PATH = ArcGetPath(#OnTheFlyArcOn, WDAT1) DELAY = ArcGetDelay(#GasPreflow, WDAT1) DO ArcMainNG(#GasPreflow, WDAT1, WP3) PRIO = -1
  TRIGGER WHEN PATH = ArcGetPath(#OnTheFlyArcOn, WDAT1) DELAY = 0 DO ArcMainNG(#ArcOnMoveStd, WDAT1, WP3) PRIO = -1
  ArcMainNG(#ArcOnBeforeMoveStd, WDAT1, WP3)
  LIN XP3
  ArcMainNG(#ArcOnAfterMoveStd, WDAT1, WP3)
;ENDFOLD
   $VEL.CP = 0.025
   LIN  {X -9.800, Y 9.800, Z 0.300, A 0.000, B 0.000, C 0.000} C_DIS
   $VEL.CP = 0.030
   LIN  {X -9.800, Y -9.800, Z 0.300, A 0.000, B 0.000, C 0.000} C_DIS
   $VEL.CP = 0.030
   LIN  {X 9.800, Y -9.800, Z 0.300, A 0.000, B 0.000, C 0.000} C_DIS
   $VEL.CP = 0.030
   LIN  {X 9.800, Y 9.800, Z 0.300, A 0.000, B 0.000, C 0.000} C_DIS
   $VEL.CP = 0.030
   LIN  {X -9.800, Y 9.800, Z 0.300, A 0.000, B 0.000, C 0.000} C_DIS

;FOLD ARCOFF WDAT2 LIN P4 CPDAT2 Tool[1]:cmttorch Base[1]:vrashatel ;%{PE}
  ;FOLD Parameters ;%{h}
    ;Params IlfProvider=kukaroboter.arctech.arcofflin; Kuka.IsGlobalPoint=False; Kuka.PointName=P4; Kuka.BlendingEnabled=False; Kuka.MoveDataName=CPDAT2; Kuka.VelocityPath=0.01; Kuka.CurrentCDSetIndex=0; Kuka.MovementParameterFieldEnabled=True; ArcTech.WdatVarName=WDAT2; ArcTech.Basic=3.4.3.1264
  ;ENDFOLD
  $BWDSTART = FALSE
  LDAT_ACT = LCPDAT2
  FDAT_ACT = FP4
  BAS(#CP_PARAMS, gArcBasVelDefinition)
  SET_CD_PARAMS (0)
  TRIGGER WHEN PATH = ArcGetPath(#ArcOffBefore, WDAT2) DELAY = 0 DO ArcMainNG(#ArcOffBeforeOffStd, WDAT2, WP4) PRIO = -1
  TRIGGER WHEN PATH = ArcGetPath(#OnTheFlyArcOff, WDAT2) DELAY = 0 DO ArcMainNG(#ArcOffMoveStd, WDAT2, WP4) PRIO = -1
  ArcMainNG(#ArcOffBeforeMoveStd, WDAT2, WP4)
  LIN XP4
  ArcMainNG(#ArcOffAfterMoveStd, WDAT2, WP4)
;ENDFOLD
   $VEL.CP = 0.030
   LIN  {X -9.800, Y 9.600, Z 0.300, A 0.000, B 0.000, C 0.000} C_DIS
   $VEL.CP = 0.030
   LIN  {X -9.360, Y 9.360, Z 0.300, A 0.000, B 0.000, C 0.000} C_DIS
   $VEL.CP = 0.030
   LIN  {X -9.400, Y 9.400, Z 0.300, A 0.000, B 0.000, C 0.000} C_DIS

;FOLD ARCON WDAT1 LIN P3 Vel=0.5 m/s CPDAT1 Tool[1]:cmttorch Base[1]:vrashatel ;%{PE}
  ;FOLD Parameters ;%{h}
    ;Params IlfProvider=kukaroboter.arctech.arconlin; Kuka.IsGlobalPoint=False; Kuka.PointName=P3; Kuka.BlendingEnabled=False; Kuka.MoveDataName=CPDAT1; Kuka.VelocityPath=0.5; Kuka.CurrentCDSetIndex=0; Kuka.MovementParameterFieldEnabled=True; ArcTech.WdatVarName=WDAT1; ArcTech.Basic=3.4.3.1264
  ;ENDFOLD
  $BWDSTART = FALSE
  LDAT_ACT = LCPDAT1
  FDAT_ACT = FP3
  BAS(#CP_PARAMS, 0.5)
  SET_CD_PARAMS (0)
  TRIGGER WHEN DISTANCE = 1 DELAY = ArcGetDelay(#PreDefinition, WDAT1) DO ArcMainNG(#PreDefinition, WDAT1, WP3) PRIO = -1
  TRIGGER WHEN PATH = ArcGetPath(#OnTheFlyArcOn, WDAT1) DELAY = ArcGetDelay(#GasPreflow, WDAT1) DO ArcMainNG(#GasPreflow, WDAT1, WP3) PRIO = -1
  TRIGGER WHEN PATH = ArcGetPath(#OnTheFlyArcOn, WDAT1) DELAY = 0 DO ArcMainNG(#ArcOnMoveStd, WDAT1, WP3) PRIO = -1
  ArcMainNG(#ArcOnBeforeMoveStd, WDAT1, WP3)
  LIN XP3
  ArcMainNG(#ArcOnAfterMoveStd, WDAT1, WP3)
;ENDFOLD
   $VEL.CP = 0.030
   LIN  {X -9.400, Y -9.400, Z 0.300, A 0.000, B 0.000, C 0.000} C_DIS
   $VEL.CP = 0.030
   LIN  {X 9.400, Y -9.400, Z 0.300, A 0.000, B 0.000, C 0.000} C_DIS
   $VEL.CP = 0.030
   LIN  {X 9.400, Y 9.400, Z 0.300, A 0.000, B 0.000, C 0.000} C_DIS
   $VEL.CP = 0.030
   LIN  {X -9.400, Y 9.400, Z 0.300, A 0.000, B 0.000, C 0.000} C_DIS

;FOLD ARCOFF WDAT2 LIN P4 CPDAT2 Tool[1]:cmttorch Base[1]:vrashatel ;%{PE}
  ;FOLD Parameters ;%{h}
    ;Params IlfProvider=kukaroboter.arctech.arcofflin; Kuka.IsGlobalPoint=False; Kuka.PointName=P4; Kuka.BlendingEnabled=False; Kuka.MoveDataName=CPDAT2; Kuka.VelocityPath=0.01; Kuka.CurrentCDSetIndex=0; Kuka.MovementParameterFieldEnabled=True; ArcTech.WdatVarName=WDAT2; ArcTech.Basic=3.4.3.1264
  ;ENDFOLD
  $BWDSTART = FALSE
  LDAT_ACT = LCPDAT2
  FDAT_ACT = FP4
  BAS(#CP_PARAMS, gArcBasVelDefinition)
  SET_CD_PARAMS (0)
  TRIGGER WHEN PATH = ArcGetPath(#ArcOffBefore, WDAT2) DELAY = 0 DO ArcMainNG(#ArcOffBeforeOffStd, WDAT2, WP4) PRIO = -1
  TRIGGER WHEN PATH = ArcGetPath(#OnTheFlyArcOff, WDAT2) DELAY = 0 DO ArcMainNG(#ArcOffMoveStd, WDAT2, WP4) PRIO = -1
  ArcMainNG(#ArcOffBeforeMoveStd, WDAT2, WP4)
  LIN XP4
  ArcMainNG(#ArcOffAfterMoveStd, WDAT2, WP4)
;ENDFOLD
   $VEL.CP = 0.030
   LIN  {X -9.010, Y 9.010, Z 0.300, A 0.000, B 0.000, C 0.000} C_DIS

;FOLD ARCON WDAT1 LIN P3 Vel=0.5 m/s CPDAT1 Tool[1]:cmttorch Base[1]:vrashatel ;%{PE}
  ;FOLD Parameters ;%{h}
    ;Params IlfProvider=kukaroboter.arctech.arconlin; Kuka.IsGlobalPoint=False; Kuka.PointName=P3; Kuka.BlendingEnabled=False; Kuka.MoveDataName=CPDAT1; Kuka.VelocityPath=0.5; Kuka.CurrentCDSetIndex=0; Kuka.MovementParameterFieldEnabled=True; ArcTech.WdatVarName=WDAT1; ArcTech.Basic=3.4.3.1264
  ;ENDFOLD
  $BWDSTART = FALSE
  LDAT_ACT = LCPDAT1
  FDAT_ACT = FP3
  BAS(#CP_PARAMS, 0.5)
  SET_CD_PARAMS (0)
  TRIGGER WHEN DISTANCE = 1 DELAY = ArcGetDelay(#PreDefinition, WDAT1) DO ArcMainNG(#PreDefinition, WDAT1, WP3) PRIO = -1
  TRIGGER WHEN PATH = ArcGetPath(#OnTheFlyArcOn, WDAT1) DELAY = ArcGetDelay(#GasPreflow, WDAT1) DO ArcMainNG(#GasPreflow, WDAT1, WP3) PRIO = -1
  TRIGGER WHEN PATH = ArcGetPath(#OnTheFlyArcOn, WDAT1) DELAY = 0 DO ArcMainNG(#ArcOnMoveStd, WDAT1, WP3) PRIO = -1
  ArcMainNG(#ArcOnBeforeMoveStd, WDAT1, WP3)
  LIN XP3
  ArcMainNG(#ArcOnAfterMoveStd, WDAT1, WP3)
;ENDFOLD
   $VEL.CP = 0.030
   LIN  {X -9.010, Y -9.010, Z 0.300, A 0.000, B 0.000, C 0.000} C_DIS
   $VEL.CP = 0.030
   LIN  {X 9.010, Y -9.010, Z 0.300, A 0.000, B 0.000, C 0.000} C_DIS
   $VEL.CP = 0.030
   LIN  {X 9.010, Y 9.010, Z 0.300, A 0.000, B 0.000, C 0.000} C_DIS
   $VEL.CP = 0.030
   LIN  {X -9.010, Y 9.010, Z 0.300, A 0.000, B 0.000, C 0.000} C_DIS

;FOLD ARCOFF WDAT2 LIN P4 CPDAT2 Tool[1]:cmttorch Base[1]:vrashatel ;%{PE}
  ;FOLD Parameters ;%{h}
    ;Params IlfProvider=kukaroboter.arctech.arcofflin; Kuka.IsGlobalPoint=False; Kuka.PointName=P4; Kuka.BlendingEnabled=False; Kuka.MoveDataName=CPDAT2; Kuka.VelocityPath=0.01; Kuka.CurrentCDSetIndex=0; Kuka.MovementParameterFieldEnabled=True; ArcTech.WdatVarName=WDAT2; ArcTech.Basic=3.4.3.1264
  ;ENDFOLD
  $BWDSTART = FALSE
  LDAT_ACT = LCPDAT2
  FDAT_ACT = FP4
  BAS(#CP_PARAMS, gArcBasVelDefinition)
  SET_CD_PARAMS (0)
  TRIGGER WHEN PATH = ArcGetPath(#ArcOffBefore, WDAT2) DELAY = 0 DO ArcMainNG(#ArcOffBeforeOffStd, WDAT2, WP4) PRIO = -1
  TRIGGER WHEN PATH = ArcGetPath(#OnTheFlyArcOff, WDAT2) DELAY = 0 DO ArcMainNG(#ArcOffMoveStd, WDAT2, WP4) PRIO = -1
  ArcMainNG(#ArcOffBeforeMoveStd, WDAT2, WP4)
  LIN XP4
  ArcMainNG(#ArcOffAfterMoveStd, WDAT2, WP4)
;ENDFOLD
   $VEL.CP = 0.030
   LIN  {X -8.829, Y 8.706, Z 0.300, A 0.000, B 0.000, C 0.000} C_DIS

;FOLD ARCON WDAT1 LIN P3 Vel=0.5 m/s CPDAT1 Tool[1]:cmttorch Base[1]:vrashatel ;%{PE}
  ;FOLD Parameters ;%{h}
    ;Params IlfProvider=kukaroboter.arctech.arconlin; Kuka.IsGlobalPoint=False; Kuka.PointName=P3; Kuka.BlendingEnabled=False; Kuka.MoveDataName=CPDAT1; Kuka.VelocityPath=0.5; Kuka.CurrentCDSetIndex=0; Kuka.MovementParameterFieldEnabled=True; ArcTech.WdatVarName=WDAT1; ArcTech.Basic=3.4.3.1264
  ;ENDFOLD
  $BWDSTART = FALSE
  LDAT_ACT = LCPDAT1
  FDAT_ACT = FP3
  BAS(#CP_PARAMS, 0.5)
  SET_CD_PARAMS (0)
  TRIGGER WHEN DISTANCE = 1 DELAY = ArcGetDelay(#PreDefinition, WDAT1) DO ArcMainNG(#PreDefinition, WDAT1, WP3) PRIO = -1
  TRIGGER WHEN PATH = ArcGetPath(#OnTheFlyArcOn, WDAT1) DELAY = ArcGetDelay(#GasPreflow, WDAT1) DO ArcMainNG(#GasPreflow, WDAT1, WP3) PRIO = -1
  TRIGGER WHEN PATH = ArcGetPath(#OnTheFlyArcOn, WDAT1) DELAY = 0 DO ArcMainNG(#ArcOnMoveStd, WDAT1, WP3) PRIO = -1
  ArcMainNG(#ArcOnBeforeMoveStd, WDAT1, WP3)
  LIN XP3
  ArcMainNG(#ArcOnAfterMoveStd, WDAT1, WP3)
;ENDFOLD
   $VEL.CP = 0.030
   LIN  {X -8.706, Y 8.829, Z 0.300, A 0.000, B 0.000, C 0.000} C_DIS

;FOLD ARCOFF WDAT2 LIN P4 CPDAT2 Tool[1]:cmttorch Base[1]:vrashatel ;%{PE}
  ;FOLD Parameters ;%{h}
    ;Params IlfProvider=kukaroboter.arctech.arcofflin; Kuka.IsGlobalPoint=False; Kuka.PointName=P4; Kuka.BlendingEnabled=False; Kuka.MoveDataName=CPDAT2; Kuka.VelocityPath=0.01; Kuka.CurrentCDSetIndex=0; Kuka.MovementParameterFieldEnabled=True; ArcTech.WdatVarName=WDAT2; ArcTech.Basic=3.4.3.1264
  ;ENDFOLD
  $BWDSTART = FALSE
  LDAT_ACT = LCPDAT2
  FDAT_ACT = FP4
  BAS(#CP_PARAMS, gArcBasVelDefinition)
  SET_CD_PARAMS (0)
  TRIGGER WHEN PATH = ArcGetPath(#ArcOffBefore, WDAT2) DELAY = 0 DO ArcMainNG(#ArcOffBeforeOffStd, WDAT2, WP4) PRIO = -1
  TRIGGER WHEN PATH = ArcGetPath(#OnTheFlyArcOff, WDAT2) DELAY = 0 DO ArcMainNG(#ArcOffMoveStd, WDAT2, WP4) PRIO = -1
  ArcMainNG(#ArcOffBeforeMoveStd, WDAT2, WP4)
  LIN XP4
  ArcMainNG(#ArcOffAfterMoveStd, WDAT2, WP4)
;ENDFOLD
   $VEL.CP = 0.030
   LIN  {X -8.140, Y 8.829, Z 0.300, A 0.000, B 0.000, C 0.000} C_DIS

;FOLD ARCON WDAT1 LIN P3 Vel=0.5 m/s CPDAT1 Tool[1]:cmttorch Base[1]:vrashatel ;%{PE}
  ;FOLD Parameters ;%{h}
    ;Params IlfProvider=kukaroboter.arctech.arconlin; Kuka.IsGlobalPoint=False; Kuka.PointName=P3; Kuka.BlendingEnabled=False; Kuka.MoveDataName=CPDAT1; Kuka.VelocityPath=0.5; Kuka.CurrentCDSetIndex=0; Kuka.MovementParameterFieldEnabled=True; ArcTech.WdatVarName=WDAT1; ArcTech.Basic=3.4.3.1264
  ;ENDFOLD
  $BWDSTART = FALSE
  LDAT_ACT = LCPDAT1
  FDAT_ACT = FP3
  BAS(#CP_PARAMS, 0.5)
  SET_CD_PARAMS (0)
  TRIGGER WHEN DISTANCE = 1 DELAY = ArcGetDelay(#PreDefinition, WDAT1) DO ArcMainNG(#PreDefinition, WDAT1, WP3) PRIO = -1
  TRIGGER WHEN PATH = ArcGetPath(#OnTheFlyArcOn, WDAT1) DELAY = ArcGetDelay(#GasPreflow, WDAT1) DO ArcMainNG(#GasPreflow, WDAT1, WP3) PRIO = -1
  TRIGGER WHEN PATH = ArcGetPath(#OnTheFlyArcOn, WDAT1) DELAY = 0 DO ArcMainNG(#ArcOnMoveStd, WDAT1, WP3) PRIO = -1
  ArcMainNG(#ArcOnBeforeMoveStd, WDAT1, WP3)
  LIN XP3
  ArcMainNG(#ArcOnAfterMoveStd, WDAT1, WP3)
;ENDFOLD
   $VEL.CP = 0.030
   LIN  {X -8.829, Y 8.140, Z 0.300, A 0.000, B 0.000, C 0.000} C_DIS

;FOLD ARCOFF WDAT2 LIN P4 CPDAT2 Tool[1]:cmttorch Base[1]:vrashatel ;%{PE}
  ;FOLD Parameters ;%{h}
    ;Params IlfProvider=kukaroboter.arctech.arcofflin; Kuka.IsGlobalPoint=False; Kuka.PointName=P4; Kuka.BlendingEnabled=False; Kuka.MoveDataName=CPDAT2; Kuka.VelocityPath=0.01; Kuka.CurrentCDSetIndex=0; Kuka.MovementParameterFieldEnabled=True; ArcTech.WdatVarName=WDAT2; ArcTech.Basic=3.4.3.1264
  ;ENDFOLD
  $BWDSTART = FALSE
  LDAT_ACT = LCPDAT2
  FDAT_ACT = FP4
  BAS(#CP_PARAMS, gArcBasVelDefinition)
  SET_CD_PARAMS (0)
  TRIGGER WHEN PATH = ArcGetPath(#ArcOffBefore, WDAT2) DELAY = 0 DO ArcMainNG(#ArcOffBeforeOffStd, WDAT2, WP4) PRIO = -1
  TRIGGER WHEN PATH = ArcGetPath(#OnTheFlyArcOff, WDAT2) DELAY = 0 DO ArcMainNG(#ArcOffMoveStd, WDAT2, WP4) PRIO = -1
  ArcMainNG(#ArcOffBeforeMoveStd, WDAT2, WP4)
  LIN XP4
  ArcMainNG(#ArcOffAfterMoveStd, WDAT2, WP4)
;ENDFOLD
   $VEL.CP = 0.030
   LIN  {X -8.829, Y 7.575, Z 0.300, A 0.000, B 0.000, C 0.000} C_DIS

;FOLD ARCON WDAT1 LIN P3 Vel=0.5 m/s CPDAT1 Tool[1]:cmttorch Base[1]:vrashatel ;%{PE}
  ;FOLD Parameters ;%{h}
    ;Params IlfProvider=kukaroboter.arctech.arconlin; Kuka.IsGlobalPoint=False; Kuka.PointName=P3; Kuka.BlendingEnabled=False; Kuka.MoveDataName=CPDAT1; Kuka.VelocityPath=0.5; Kuka.CurrentCDSetIndex=0; Kuka.MovementParameterFieldEnabled=True; ArcTech.WdatVarName=WDAT1; ArcTech.Basic=3.4.3.1264
  ;ENDFOLD
  $BWDSTART = FALSE
  LDAT_ACT = LCPDAT1
  FDAT_ACT = FP3
  BAS(#CP_PARAMS, 0.5)
  SET_CD_PARAMS (0)
  TRIGGER WHEN DISTANCE = 1 DELAY = ArcGetDelay(#PreDefinition, WDAT1) DO ArcMainNG(#PreDefinition, WDAT1, WP3) PRIO = -1
  TRIGGER WHEN PATH = ArcGetPath(#OnTheFlyArcOn, WDAT1) DELAY = ArcGetDelay(#GasPreflow, WDAT1) DO ArcMainNG(#GasPreflow, WDAT1, WP3) PRIO = -1
  TRIGGER WHEN PATH = ArcGetPath(#OnTheFlyArcOn, WDAT1) DELAY = 0 DO ArcMainNG(#ArcOnMoveStd, WDAT1, WP3) PRIO = -1
  ArcMainNG(#ArcOnBeforeMoveStd, WDAT1, WP3)
  LIN XP3
  ArcMainNG(#ArcOnAfterMoveStd, WDAT1, WP3)
;ENDFOLD
   $VEL.CP = 0.030
   LIN  {X -7.575, Y 8.829, Z 0.300, A 0.000, B 0.000, C 0.000} C_DIS

;FOLD ARCOFF WDAT2 LIN P4 CPDAT2 Tool[1]:cmttorch Base[1]:vrashatel ;%{PE}
  ;FOLD Parameters ;%{h}
    ;Params IlfProvider=kukaroboter.arctech.arcofflin; Kuka.IsGlobalPoint=False; Kuka.PointName=P4; Kuka.BlendingEnabled=False; Kuka.MoveDataName=CPDAT2; Kuka.VelocityPath=0.01; Kuka.CurrentCDSetIndex=0; Kuka.MovementParameterFieldEnabled=True; ArcTech.WdatVarName=WDAT2; ArcTech.Basic=3.4.3.1264
  ;ENDFOLD
  $BWDSTART = FALSE
  LDAT_ACT = LCPDAT2
  FDAT_ACT = FP4
  BAS(#CP_PARAMS, gArcBasVelDefinition)
  SET_CD_PARAMS (0)
  TRIGGER WHEN PATH = ArcGetPath(#ArcOffBefore, WDAT2) DELAY = 0 DO ArcMainNG(#ArcOffBeforeOffStd, WDAT2, WP4) PRIO = -1
  TRIGGER WHEN PATH = ArcGetPath(#OnTheFlyArcOff, WDAT2) DELAY = 0 DO ArcMainNG(#ArcOffMoveStd, WDAT2, WP4) PRIO = -1
  ArcMainNG(#ArcOffBeforeMoveStd, WDAT2, WP4)
  LIN XP4
  ArcMainNG(#ArcOffAfterMoveStd, WDAT2, WP4)
;ENDFOLD
   $VEL.CP = 0.030
   LIN  {X -7.009, Y 8.829, Z 0.300, A 0.000, B 0.000, C 0.000} C_DIS

;FOLD ARCON WDAT1 LIN P3 Vel=0.5 m/s CPDAT1 Tool[1]:cmttorch Base[1]:vrashatel ;%{PE}
  ;FOLD Parameters ;%{h}
    ;Params IlfProvider=kukaroboter.arctech.arconlin; Kuka.IsGlobalPoint=False; Kuka.PointName=P3; Kuka.BlendingEnabled=False; Kuka.MoveDataName=CPDAT1; Kuka.VelocityPath=0.5; Kuka.CurrentCDSetIndex=0; Kuka.MovementParameterFieldEnabled=True; ArcTech.WdatVarName=WDAT1; ArcTech.Basic=3.4.3.1264
  ;ENDFOLD
  $BWDSTART = FALSE
  LDAT_ACT = LCPDAT1
  FDAT_ACT = FP3
  BAS(#CP_PARAMS, 0.5)
  SET_CD_PARAMS (0)
  TRIGGER WHEN DISTANCE = 1 DELAY = ArcGetDelay(#PreDefinition, WDAT1) DO ArcMainNG(#PreDefinition, WDAT1, WP3) PRIO = -1
  TRIGGER WHEN PATH = ArcGetPath(#OnTheFlyArcOn, WDAT1) DELAY = ArcGetDelay(#GasPreflow, WDAT1) DO ArcMainNG(#GasPreflow, WDAT1, WP3) PRIO = -1
  TRIGGER WHEN PATH = ArcGetPath(#OnTheFlyArcOn, WDAT1) DELAY = 0 DO ArcMainNG(#ArcOnMoveStd, WDAT1, WP3) PRIO = -1
  ArcMainNG(#ArcOnBeforeMoveStd, WDAT1, WP3)
  LIN XP3
  ArcMainNG(#ArcOnAfterMoveStd, WDAT1, WP3)
;ENDFOLD
   $VEL.CP = 0.030
   LIN  {X -8.829, Y 7.009, Z 0.300, A 0.000, B 0.000, C 0.000} C_DIS

;FOLD ARCOFF WDAT2 LIN P4 CPDAT2 Tool[1]:cmttorch Base[1]:vrashatel ;%{PE}
  ;FOLD Parameters ;%{h}
    ;Params IlfProvider=kukaroboter.arctech.arcofflin; Kuka.IsGlobalPoint=False; Kuka.PointName=P4; Kuka.BlendingEnabled=False; Kuka.MoveDataName=CPDAT2; Kuka.VelocityPath=0.01; Kuka.CurrentCDSetIndex=0; Kuka.MovementParameterFieldEnabled=True; ArcTech.WdatVarName=WDAT2; ArcTech.Basic=3.4.3.1264
  ;ENDFOLD
  $BWDSTART = FALSE
  LDAT_ACT = LCPDAT2
  FDAT_ACT = FP4
  BAS(#CP_PARAMS, gArcBasVelDefinition)
  SET_CD_PARAMS (0)
  TRIGGER WHEN PATH = ArcGetPath(#ArcOffBefore, WDAT2) DELAY = 0 DO ArcMainNG(#ArcOffBeforeOffStd, WDAT2, WP4) PRIO = -1
  TRIGGER WHEN PATH = ArcGetPath(#OnTheFlyArcOff, WDAT2) DELAY = 0 DO ArcMainNG(#ArcOffMoveStd, WDAT2, WP4) PRIO = -1
  ArcMainNG(#ArcOffBeforeMoveStd, WDAT2, WP4)
  LIN XP4
  ArcMainNG(#ArcOffAfterMoveStd, WDAT2, WP4)
;ENDFOLD
   $VEL.CP = 0.030
   LIN  {X -8.829, Y 6.443, Z 0.300, A 0.000, B 0.000, C 0.000} C_DIS

;FOLD ARCON WDAT1 LIN P3 Vel=0.5 m/s CPDAT1 Tool[1]:cmttorch Base[1]:vrashatel ;%{PE}
  ;FOLD Parameters ;%{h}
    ;Params IlfProvider=kukaroboter.arctech.arconlin; Kuka.IsGlobalPoint=False; Kuka.PointName=P3; Kuka.BlendingEnabled=False; Kuka.MoveDataName=CPDAT1; Kuka.VelocityPath=0.5; Kuka.CurrentCDSetIndex=0; Kuka.MovementParameterFieldEnabled=True; ArcTech.WdatVarName=WDAT1; ArcTech.Basic=3.4.3.1264
  ;ENDFOLD
  $BWDSTART = FALSE
  LDAT_ACT = LCPDAT1
  FDAT_ACT = FP3
  BAS(#CP_PARAMS, 0.5)
  SET_CD_PARAMS (0)
  TRIGGER WHEN DISTANCE = 1 DELAY = ArcGetDelay(#PreDefinition, WDAT1) DO ArcMainNG(#PreDefinition, WDAT1, WP3) PRIO = -1
  TRIGGER WHEN PATH = ArcGetPath(#OnTheFlyArcOn, WDAT1) DELAY = ArcGetDelay(#GasPreflow, WDAT1) DO ArcMainNG(#GasPreflow, WDAT1, WP3) PRIO = -1
  TRIGGER WHEN PATH = ArcGetPath(#OnTheFlyArcOn, WDAT1) DELAY = 0 DO ArcMainNG(#ArcOnMoveStd, WDAT1, WP3) PRIO = -1
  ArcMainNG(#ArcOnBeforeMoveStd, WDAT1, WP3)
  LIN XP3
  ArcMainNG(#ArcOnAfterMoveStd, WDAT1, WP3)
;ENDFOLD
   $VEL.CP = 0.030
   LIN  {X -6.443, Y 8.829, Z 0.300, A 0.000, B 0.000, C 0.000} C_DIS

;FOLD ARCOFF WDAT2 LIN P4 CPDAT2 Tool[1]:cmttorch Base[1]:vrashatel ;%{PE}
  ;FOLD Parameters ;%{h}
    ;Params IlfProvider=kukaroboter.arctech.arcofflin; Kuka.IsGlobalPoint=False; Kuka.PointName=P4; Kuka.BlendingEnabled=False; Kuka.MoveDataName=CPDAT2; Kuka.VelocityPath=0.01; Kuka.CurrentCDSetIndex=0; Kuka.MovementParameterFieldEnabled=True; ArcTech.WdatVarName=WDAT2; ArcTech.Basic=3.4.3.1264
  ;ENDFOLD
  $BWDSTART = FALSE
  LDAT_ACT = LCPDAT2
  FDAT_ACT = FP4
  BAS(#CP_PARAMS, gArcBasVelDefinition)
  SET_CD_PARAMS (0)
  TRIGGER WHEN PATH = ArcGetPath(#ArcOffBefore, WDAT2) DELAY = 0 DO ArcMainNG(#ArcOffBeforeOffStd, WDAT2, WP4) PRIO = -1
  TRIGGER WHEN PATH = ArcGetPath(#OnTheFlyArcOff, WDAT2) DELAY = 0 DO ArcMainNG(#ArcOffMoveStd, WDAT2, WP4) PRIO = -1
  ArcMainNG(#ArcOffBeforeMoveStd, WDAT2, WP4)
  LIN XP4
  ArcMainNG(#ArcOffAfterMoveStd, WDAT2, WP4)
;ENDFOLD
   $VEL.CP = 0.030
   LIN  {X -5.878, Y 8.829, Z 0.300, A 0.000, B 0.000, C 0.000} C_DIS

;FOLD ARCON WDAT1 LIN P3 Vel=0.5 m/s CPDAT1 Tool[1]:cmttorch Base[1]:vrashatel ;%{PE}
  ;FOLD Parameters ;%{h}
    ;Params IlfProvider=kukaroboter.arctech.arconlin; Kuka.IsGlobalPoint=False; Kuka.PointName=P3; Kuka.BlendingEnabled=False; Kuka.MoveDataName=CPDAT1; Kuka.VelocityPath=0.5; Kuka.CurrentCDSetIndex=0; Kuka.MovementParameterFieldEnabled=True; ArcTech.WdatVarName=WDAT1; ArcTech.Basic=3.4.3.1264
  ;ENDFOLD
  $BWDSTART = FALSE
  LDAT_ACT = LCPDAT1
  FDAT_ACT = FP3
  BAS(#CP_PARAMS, 0.5)
  SET_CD_PARAMS (0)
  TRIGGER WHEN DISTANCE = 1 DELAY = ArcGetDelay(#PreDefinition, WDAT1) DO ArcMainNG(#PreDefinition, WDAT1, WP3) PRIO = -1
  TRIGGER WHEN PATH = ArcGetPath(#OnTheFlyArcOn, WDAT1) DELAY = ArcGetDelay(#GasPreflow, WDAT1) DO ArcMainNG(#GasPreflow, WDAT1, WP3) PRIO = -1
  TRIGGER WHEN PATH = ArcGetPath(#OnTheFlyArcOn, WDAT1) DELAY = 0 DO ArcMainNG(#ArcOnMoveStd, WDAT1, WP3) PRIO = -1
  ArcMainNG(#ArcOnBeforeMoveStd, WDAT1, WP3)
  LIN XP3
  ArcMainNG(#ArcOnAfterMoveStd, WDAT1, WP3)
;ENDFOLD
   $VEL.CP = 0.030
   LIN  {X -8.829, Y 5.878, Z 0.300, A 0.000, B 0.000, C 0.000} C_DIS

;FOLD ARCOFF WDAT2 LIN P4 CPDAT2 Tool[1]:cmttorch Base[1]:vrashatel ;%{PE}
  ;FOLD Parameters ;%{h}
    ;Params IlfProvider=kukaroboter.arctech.arcofflin; Kuka.IsGlobalPoint=False; Kuka.PointName=P4; Kuka.BlendingEnabled=False; Kuka.MoveDataName=CPDAT2; Kuka.VelocityPath=0.01; Kuka.CurrentCDSetIndex=0; Kuka.MovementParameterFieldEnabled=True; ArcTech.WdatVarName=WDAT2; ArcTech.Basic=3.4.3.1264
  ;ENDFOLD
  $BWDSTART = FALSE
  LDAT_ACT = LCPDAT2
  FDAT_ACT = FP4
  BAS(#CP_PARAMS, gArcBasVelDefinition)
  SET_CD_PARAMS (0)
  TRIGGER WHEN PATH = ArcGetPath(#ArcOffBefore, WDAT2) DELAY = 0 DO ArcMainNG(#ArcOffBeforeOffStd, WDAT2, WP4) PRIO = -1
  TRIGGER WHEN PATH = ArcGetPath(#OnTheFlyArcOff, WDAT2) DELAY = 0 DO ArcMainNG(#ArcOffMoveStd, WDAT2, WP4) PRIO = -1
  ArcMainNG(#ArcOffBeforeMoveStd, WDAT2, WP4)
  LIN XP4
  ArcMainNG(#ArcOffAfterMoveStd, WDAT2, WP4)
;ENDFOLD
   $VEL.CP = 0.030
   LIN  {X -8.829, Y 5.312, Z 0.300, A 0.000, B 0.000, C 0.000} C_DIS

;FOLD ARCON WDAT1 LIN P3 Vel=0.5 m/s CPDAT1 Tool[1]:cmttorch Base[1]:vrashatel ;%{PE}
  ;FOLD Parameters ;%{h}
    ;Params IlfProvider=kukaroboter.arctech.arconlin; Kuka.IsGlobalPoint=False; Kuka.PointName=P3; Kuka.BlendingEnabled=False; Kuka.MoveDataName=CPDAT1; Kuka.VelocityPath=0.5; Kuka.CurrentCDSetIndex=0; Kuka.MovementParameterFieldEnabled=True; ArcTech.WdatVarName=WDAT1; ArcTech.Basic=3.4.3.1264
  ;ENDFOLD
  $BWDSTART = FALSE
  LDAT_ACT = LCPDAT1
  FDAT_ACT = FP3
  BAS(#CP_PARAMS, 0.5)
  SET_CD_PARAMS (0)
  TRIGGER WHEN DISTANCE = 1 DELAY = ArcGetDelay(#PreDefinition, WDAT1) DO ArcMainNG(#PreDefinition, WDAT1, WP3) PRIO = -1
  TRIGGER WHEN PATH = ArcGetPath(#OnTheFlyArcOn, WDAT1) DELAY = ArcGetDelay(#GasPreflow, WDAT1) DO ArcMainNG(#GasPreflow, WDAT1, WP3) PRIO = -1
  TRIGGER WHEN PATH = ArcGetPath(#OnTheFlyArcOn, WDAT1) DELAY = 0 DO ArcMainNG(#ArcOnMoveStd, WDAT1, WP3) PRIO = -1
  ArcMainNG(#ArcOnBeforeMoveStd, WDAT1, WP3)
  LIN XP3
  ArcMainNG(#ArcOnAfterMoveStd, WDAT1, WP3)
;ENDFOLD
   $VEL.CP = 0.030
   LIN  {X -5.312, Y 8.829, Z 0.300, A 0.000, B 0.000, C 0.000} C_DIS

;FOLD ARCOFF WDAT2 LIN P4 CPDAT2 Tool[1]:cmttorch Base[1]:vrashatel ;%{PE}
  ;FOLD Parameters ;%{h}
    ;Params IlfProvider=kukaroboter.arctech.arcofflin; Kuka.IsGlobalPoint=False; Kuka.PointName=P4; Kuka.BlendingEnabled=False; Kuka.MoveDataName=CPDAT2; Kuka.VelocityPath=0.01; Kuka.CurrentCDSetIndex=0; Kuka.MovementParameterFieldEnabled=True; ArcTech.WdatVarName=WDAT2; ArcTech.Basic=3.4.3.1264
  ;ENDFOLD
  $BWDSTART = FALSE
  LDAT_ACT = LCPDAT2
  FDAT_ACT = FP4
  BAS(#CP_PARAMS, gArcBasVelDefinition)
  SET_CD_PARAMS (0)
  TRIGGER WHEN PATH = ArcGetPath(#ArcOffBefore, WDAT2) DELAY = 0 DO ArcMainNG(#ArcOffBeforeOffStd, WDAT2, WP4) PRIO = -1
  TRIGGER WHEN PATH = ArcGetPath(#OnTheFlyArcOff, WDAT2) DELAY = 0 DO ArcMainNG(#ArcOffMoveStd, WDAT2, WP4) PRIO = -1
  ArcMainNG(#ArcOffBeforeMoveStd, WDAT2, WP4)
  LIN XP4
  ArcMainNG(#ArcOffAfterMoveStd, WDAT2, WP4)
;ENDFOLD
   $VEL.CP = 0.030
   LIN  {X -4.746, Y 8.829, Z 0.300, A 0.000, B 0.000, C 0.000} C_DIS

;FOLD ARCON WDAT1 LIN P3 Vel=0.5 m/s CPDAT1 Tool[1]:cmttorch Base[1]:vrashatel ;%{PE}
  ;FOLD Parameters ;%{h}
    ;Params IlfProvider=kukaroboter.arctech.arconlin; Kuka.IsGlobalPoint=False; Kuka.PointName=P3; Kuka.BlendingEnabled=False; Kuka.MoveDataName=CPDAT1; Kuka.VelocityPath=0.5; Kuka.CurrentCDSetIndex=0; Kuka.MovementParameterFieldEnabled=True; ArcTech.WdatVarName=WDAT1; ArcTech.Basic=3.4.3.1264
  ;ENDFOLD
  $BWDSTART = FALSE
  LDAT_ACT = LCPDAT1
  FDAT_ACT = FP3
  BAS(#CP_PARAMS, 0.5)
  SET_CD_PARAMS (0)
  TRIGGER WHEN DISTANCE = 1 DELAY = ArcGetDelay(#PreDefinition, WDAT1) DO ArcMainNG(#PreDefinition, WDAT1, WP3) PRIO = -1
  TRIGGER WHEN PATH = ArcGetPath(#OnTheFlyArcOn, WDAT1) DELAY = ArcGetDelay(#GasPreflow, WDAT1) DO ArcMainNG(#GasPreflow, WDAT1, WP3) PRIO = -1
  TRIGGER WHEN PATH = ArcGetPath(#OnTheFlyArcOn, WDAT1) DELAY = 0 DO ArcMainNG(#ArcOnMoveStd, WDAT1, WP3) PRIO = -1
  ArcMainNG(#ArcOnBeforeMoveStd, WDAT1, WP3)
  LIN XP3
  ArcMainNG(#ArcOnAfterMoveStd, WDAT1, WP3)
;ENDFOLD
   $VEL.CP = 0.030
   LIN  {X -8.829, Y 4.746, Z 0.300, A 0.000, B 0.000, C 0.000} C_DIS

;FOLD ARCOFF WDAT2 LIN P4 CPDAT2 Tool[1]:cmttorch Base[1]:vrashatel ;%{PE}
  ;FOLD Parameters ;%{h}
    ;Params IlfProvider=kukaroboter.arctech.arcofflin; Kuka.IsGlobalPoint=False; Kuka.PointName=P4; Kuka.BlendingEnabled=False; Kuka.MoveDataName=CPDAT2; Kuka.VelocityPath=0.01; Kuka.CurrentCDSetIndex=0; Kuka.MovementParameterFieldEnabled=True; ArcTech.WdatVarName=WDAT2; ArcTech.Basic=3.4.3.1264
  ;ENDFOLD
  $BWDSTART = FALSE
  LDAT_ACT = LCPDAT2
  FDAT_ACT = FP4
  BAS(#CP_PARAMS, gArcBasVelDefinition)
  SET_CD_PARAMS (0)
  TRIGGER WHEN PATH = ArcGetPath(#ArcOffBefore, WDAT2) DELAY = 0 DO ArcMainNG(#ArcOffBeforeOffStd, WDAT2, WP4) PRIO = -1
  TRIGGER WHEN PATH = ArcGetPath(#OnTheFlyArcOff, WDAT2) DELAY = 0 DO ArcMainNG(#ArcOffMoveStd, WDAT2, WP4) PRIO = -1
  ArcMainNG(#ArcOffBeforeMoveStd, WDAT2, WP4)
  LIN XP4
  ArcMainNG(#ArcOffAfterMoveStd, WDAT2, WP4)
;ENDFOLD
   $VEL.CP = 0.030
   LIN  {X -8.829, Y 4.181, Z 0.300, A 0.000, B 0.000, C 0.000} C_DIS

;FOLD ARCON WDAT1 LIN P3 Vel=0.5 m/s CPDAT1 Tool[1]:cmttorch Base[1]:vrashatel ;%{PE}
  ;FOLD Parameters ;%{h}
    ;Params IlfProvider=kukaroboter.arctech.arconlin; Kuka.IsGlobalPoint=False; Kuka.PointName=P3; Kuka.BlendingEnabled=False; Kuka.MoveDataName=CPDAT1; Kuka.VelocityPath=0.5; Kuka.CurrentCDSetIndex=0; Kuka.MovementParameterFieldEnabled=True; ArcTech.WdatVarName=WDAT1; ArcTech.Basic=3.4.3.1264
  ;ENDFOLD
  $BWDSTART = FALSE
  LDAT_ACT = LCPDAT1
  FDAT_ACT = FP3
  BAS(#CP_PARAMS, 0.5)
  SET_CD_PARAMS (0)
  TRIGGER WHEN DISTANCE = 1 DELAY = ArcGetDelay(#PreDefinition, WDAT1) DO ArcMainNG(#PreDefinition, WDAT1, WP3) PRIO = -1
  TRIGGER WHEN PATH = ArcGetPath(#OnTheFlyArcOn, WDAT1) DELAY = ArcGetDelay(#GasPreflow, WDAT1) DO ArcMainNG(#GasPreflow, WDAT1, WP3) PRIO = -1
  TRIGGER WHEN PATH = ArcGetPath(#OnTheFlyArcOn, WDAT1) DELAY = 0 DO ArcMainNG(#ArcOnMoveStd, WDAT1, WP3) PRIO = -1
  ArcMainNG(#ArcOnBeforeMoveStd, WDAT1, WP3)
  LIN XP3
  ArcMainNG(#ArcOnAfterMoveStd, WDAT1, WP3)
;ENDFOLD
   $VEL.CP = 0.030
   LIN  {X -4.181, Y 8.829, Z 0.300, A 0.000, B 0.000, C 0.000} C_DIS

;FOLD ARCOFF WDAT2 LIN P4 CPDAT2 Tool[1]:cmttorch Base[1]:vrashatel ;%{PE}
  ;FOLD Parameters ;%{h}
    ;Params IlfProvider=kukaroboter.arctech.arcofflin; Kuka.IsGlobalPoint=False; Kuka.PointName=P4; Kuka.BlendingEnabled=False; Kuka.MoveDataName=CPDAT2; Kuka.VelocityPath=0.01; Kuka.CurrentCDSetIndex=0; Kuka.MovementParameterFieldEnabled=True; ArcTech.WdatVarName=WDAT2; ArcTech.Basic=3.4.3.1264
  ;ENDFOLD
  $BWDSTART = FALSE
  LDAT_ACT = LCPDAT2
  FDAT_ACT = FP4
  BAS(#CP_PARAMS, gArcBasVelDefinition)
  SET_CD_PARAMS (0)
  TRIGGER WHEN PATH = ArcGetPath(#ArcOffBefore, WDAT2) DELAY = 0 DO ArcMainNG(#ArcOffBeforeOffStd, WDAT2, WP4) PRIO = -1
  TRIGGER WHEN PATH = ArcGetPath(#OnTheFlyArcOff, WDAT2) DELAY = 0 DO ArcMainNG(#ArcOffMoveStd, WDAT2, WP4) PRIO = -1
  ArcMainNG(#ArcOffBeforeMoveStd, WDAT2, WP4)
  LIN XP4
  ArcMainNG(#ArcOffAfterMoveStd, WDAT2, WP4)
;ENDFOLD
   $VEL.CP = 0.030
   LIN  {X -3.615, Y 8.829, Z 0.300, A 0.000, B 0.000, C 0.000} C_DIS

;FOLD ARCON WDAT1 LIN P3 Vel=0.5 m/s CPDAT1 Tool[1]:cmttorch Base[1]:vrashatel ;%{PE}
  ;FOLD Parameters ;%{h}
    ;Params IlfProvider=kukaroboter.arctech.arconlin; Kuka.IsGlobalPoint=False; Kuka.PointName=P3; Kuka.BlendingEnabled=False; Kuka.MoveDataName=CPDAT1; Kuka.VelocityPath=0.5; Kuka.CurrentCDSetIndex=0; Kuka.MovementParameterFieldEnabled=True; ArcTech.WdatVarName=WDAT1; ArcTech.Basic=3.4.3.1264
  ;ENDFOLD
  $BWDSTART = FALSE
  LDAT_ACT = LCPDAT1
  FDAT_ACT = FP3
  BAS(#CP_PARAMS, 0.5)
  SET_CD_PARAMS (0)
  TRIGGER WHEN DISTANCE = 1 DELAY = ArcGetDelay(#PreDefinition, WDAT1) DO ArcMainNG(#PreDefinition, WDAT1, WP3) PRIO = -1
  TRIGGER WHEN PATH = ArcGetPath(#OnTheFlyArcOn, WDAT1) DELAY = ArcGetDelay(#GasPreflow, WDAT1) DO ArcMainNG(#GasPreflow, WDAT1, WP3) PRIO = -1
  TRIGGER WHEN PATH = ArcGetPath(#OnTheFlyArcOn, WDAT1) DELAY = 0 DO ArcMainNG(#ArcOnMoveStd, WDAT1, WP3) PRIO = -1
  ArcMainNG(#ArcOnBeforeMoveStd, WDAT1, WP3)
  LIN XP3
  ArcMainNG(#ArcOnAfterMoveStd, WDAT1, WP3)
;ENDFOLD
   $VEL.CP = 0.030
   LIN  {X -8.829, Y 3.615, Z 0.300, A 0.000, B 0.000, C 0.000} C_DIS

;FOLD ARCOFF WDAT2 LIN P4 CPDAT2 Tool[1]:cmttorch Base[1]:vrashatel ;%{PE}
  ;FOLD Parameters ;%{h}
    ;Params IlfProvider=kukaroboter.arctech.arcofflin; Kuka.IsGlobalPoint=False; Kuka.PointName=P4; Kuka.BlendingEnabled=False; Kuka.MoveDataName=CPDAT2; Kuka.VelocityPath=0.01; Kuka.CurrentCDSetIndex=0; Kuka.MovementParameterFieldEnabled=True; ArcTech.WdatVarName=WDAT2; ArcTech.Basic=3.4.3.1264
  ;ENDFOLD
  $BWDSTART = FALSE
  LDAT_ACT = LCPDAT2
  FDAT_ACT = FP4
  BAS(#CP_PARAMS, gArcBasVelDefinition)
  SET_CD_PARAMS (0)
  TRIGGER WHEN PATH = ArcGetPath(#ArcOffBefore, WDAT2) DELAY = 0 DO ArcMainNG(#ArcOffBeforeOffStd, WDAT2, WP4) PRIO = -1
  TRIGGER WHEN PATH = ArcGetPath(#OnTheFlyArcOff, WDAT2) DELAY = 0 DO ArcMainNG(#ArcOffMoveStd, WDAT2, WP4) PRIO = -1
  ArcMainNG(#ArcOffBeforeMoveStd, WDAT2, WP4)
  LIN XP4
  ArcMainNG(#ArcOffAfterMoveStd, WDAT2, WP4)
;ENDFOLD
   $VEL.CP = 0.030
   LIN  {X -8.829, Y 3.049, Z 0.300, A 0.000, B 0.000, C 0.000} C_DIS

;FOLD ARCON WDAT1 LIN P3 Vel=0.5 m/s CPDAT1 Tool[1]:cmttorch Base[1]:vrashatel ;%{PE}
  ;FOLD Parameters ;%{h}
    ;Params IlfProvider=kukaroboter.arctech.arconlin; Kuka.IsGlobalPoint=False; Kuka.PointName=P3; Kuka.BlendingEnabled=False; Kuka.MoveDataName=CPDAT1; Kuka.VelocityPath=0.5; Kuka.CurrentCDSetIndex=0; Kuka.MovementParameterFieldEnabled=True; ArcTech.WdatVarName=WDAT1; ArcTech.Basic=3.4.3.1264
  ;ENDFOLD
  $BWDSTART = FALSE
  LDAT_ACT = LCPDAT1
  FDAT_ACT = FP3
  BAS(#CP_PARAMS, 0.5)
  SET_CD_PARAMS (0)
  TRIGGER WHEN DISTANCE = 1 DELAY = ArcGetDelay(#PreDefinition, WDAT1) DO ArcMainNG(#PreDefinition, WDAT1, WP3) PRIO = -1
  TRIGGER WHEN PATH = ArcGetPath(#OnTheFlyArcOn, WDAT1) DELAY = ArcGetDelay(#GasPreflow, WDAT1) DO ArcMainNG(#GasPreflow, WDAT1, WP3) PRIO = -1
  TRIGGER WHEN PATH = ArcGetPath(#OnTheFlyArcOn, WDAT1) DELAY = 0 DO ArcMainNG(#ArcOnMoveStd, WDAT1, WP3) PRIO = -1
  ArcMainNG(#ArcOnBeforeMoveStd, WDAT1, WP3)
  LIN XP3
  ArcMainNG(#ArcOnAfterMoveStd, WDAT1, WP3)
;ENDFOLD
   $VEL.CP = 0.030
   LIN  {X -3.049, Y 8.829, Z 0.300, A 0.000, B 0.000, C 0.000} C_DIS

;FOLD ARCOFF WDAT2 LIN P4 CPDAT2 Tool[1]:cmttorch Base[1]:vrashatel ;%{PE}
  ;FOLD Parameters ;%{h}
    ;Params IlfProvider=kukaroboter.arctech.arcofflin; Kuka.IsGlobalPoint=False; Kuka.PointName=P4; Kuka.BlendingEnabled=False; Kuka.MoveDataName=CPDAT2; Kuka.VelocityPath=0.01; Kuka.CurrentCDSetIndex=0; Kuka.MovementParameterFieldEnabled=True; ArcTech.WdatVarName=WDAT2; ArcTech.Basic=3.4.3.1264
  ;ENDFOLD
  $BWDSTART = FALSE
  LDAT_ACT = LCPDAT2
  FDAT_ACT = FP4
  BAS(#CP_PARAMS, gArcBasVelDefinition)
  SET_CD_PARAMS (0)
  TRIGGER WHEN PATH = ArcGetPath(#ArcOffBefore, WDAT2) DELAY = 0 DO ArcMainNG(#ArcOffBeforeOffStd, WDAT2, WP4) PRIO = -1
  TRIGGER WHEN PATH = ArcGetPath(#OnTheFlyArcOff, WDAT2) DELAY = 0 DO ArcMainNG(#ArcOffMoveStd, WDAT2, WP4) PRIO = -1
  ArcMainNG(#ArcOffBeforeMoveStd, WDAT2, WP4)
  LIN XP4
  ArcMainNG(#ArcOffAfterMoveStd, WDAT2, WP4)
;ENDFOLD
   $VEL.CP = 0.030
   LIN  {X -2.484, Y 8.829, Z 0.300, A 0.000, B 0.000, C 0.000} C_DIS

;FOLD ARCON WDAT1 LIN P3 Vel=0.5 m/s CPDAT1 Tool[1]:cmttorch Base[1]:vrashatel ;%{PE}
  ;FOLD Parameters ;%{h}
    ;Params IlfProvider=kukaroboter.arctech.arconlin; Kuka.IsGlobalPoint=False; Kuka.PointName=P3; Kuka.BlendingEnabled=False; Kuka.MoveDataName=CPDAT1; Kuka.VelocityPath=0.5; Kuka.CurrentCDSetIndex=0; Kuka.MovementParameterFieldEnabled=True; ArcTech.WdatVarName=WDAT1; ArcTech.Basic=3.4.3.1264
  ;ENDFOLD
  $BWDSTART = FALSE
  LDAT_ACT = LCPDAT1
  FDAT_ACT = FP3
  BAS(#CP_PARAMS, 0.5)
  SET_CD_PARAMS (0)
  TRIGGER WHEN DISTANCE = 1 DELAY = ArcGetDelay(#PreDefinition, WDAT1) DO ArcMainNG(#PreDefinition, WDAT1, WP3) PRIO = -1
  TRIGGER WHEN PATH = ArcGetPath(#OnTheFlyArcOn, WDAT1) DELAY = ArcGetDelay(#GasPreflow, WDAT1) DO ArcMainNG(#GasPreflow, WDAT1, WP3) PRIO = -1
  TRIGGER WHEN PATH = ArcGetPath(#OnTheFlyArcOn, WDAT1) DELAY = 0 DO ArcMainNG(#ArcOnMoveStd, WDAT1, WP3) PRIO = -1
  ArcMainNG(#ArcOnBeforeMoveStd, WDAT1, WP3)
  LIN XP3
  ArcMainNG(#ArcOnAfterMoveStd, WDAT1, WP3)
;ENDFOLD
   $VEL.CP = 0.030
   LIN  {X -8.829, Y 2.484, Z 0.300, A 0.000, B 0.000, C 0.000} C_DIS

;FOLD ARCOFF WDAT2 LIN P4 CPDAT2 Tool[1]:cmttorch Base[1]:vrashatel ;%{PE}
  ;FOLD Parameters ;%{h}
    ;Params IlfProvider=kukaroboter.arctech.arcofflin; Kuka.IsGlobalPoint=False; Kuka.PointName=P4; Kuka.BlendingEnabled=False; Kuka.MoveDataName=CPDAT2; Kuka.VelocityPath=0.01; Kuka.CurrentCDSetIndex=0; Kuka.MovementParameterFieldEnabled=True; ArcTech.WdatVarName=WDAT2; ArcTech.Basic=3.4.3.1264
  ;ENDFOLD
  $BWDSTART = FALSE
  LDAT_ACT = LCPDAT2
  FDAT_ACT = FP4
  BAS(#CP_PARAMS, gArcBasVelDefinition)
  SET_CD_PARAMS (0)
  TRIGGER WHEN PATH = ArcGetPath(#ArcOffBefore, WDAT2) DELAY = 0 DO ArcMainNG(#ArcOffBeforeOffStd, WDAT2, WP4) PRIO = -1
  TRIGGER WHEN PATH = ArcGetPath(#OnTheFlyArcOff, WDAT2) DELAY = 0 DO ArcMainNG(#ArcOffMoveStd, WDAT2, WP4) PRIO = -1
  ArcMainNG(#ArcOffBeforeMoveStd, WDAT2, WP4)
  LIN XP4
  ArcMainNG(#ArcOffAfterMoveStd, WDAT2, WP4)
;ENDFOLD
   $VEL.CP = 0.030
   LIN  {X -8.829, Y 1.918, Z 0.300, A 0.000, B 0.000, C 0.000} C_DIS

;FOLD ARCON WDAT1 LIN P3 Vel=0.5 m/s CPDAT1 Tool[1]:cmttorch Base[1]:vrashatel ;%{PE}
  ;FOLD Parameters ;%{h}
    ;Params IlfProvider=kukaroboter.arctech.arconlin; Kuka.IsGlobalPoint=False; Kuka.PointName=P3; Kuka.BlendingEnabled=False; Kuka.MoveDataName=CPDAT1; Kuka.VelocityPath=0.5; Kuka.CurrentCDSetIndex=0; Kuka.MovementParameterFieldEnabled=True; ArcTech.WdatVarName=WDAT1; ArcTech.Basic=3.4.3.1264
  ;ENDFOLD
  $BWDSTART = FALSE
  LDAT_ACT = LCPDAT1
  FDAT_ACT = FP3
  BAS(#CP_PARAMS, 0.5)
  SET_CD_PARAMS (0)
  TRIGGER WHEN DISTANCE = 1 DELAY = ArcGetDelay(#PreDefinition, WDAT1) DO ArcMainNG(#PreDefinition, WDAT1, WP3) PRIO = -1
  TRIGGER WHEN PATH = ArcGetPath(#OnTheFlyArcOn, WDAT1) DELAY = ArcGetDelay(#GasPreflow, WDAT1) DO ArcMainNG(#GasPreflow, WDAT1, WP3) PRIO = -1
  TRIGGER WHEN PATH = ArcGetPath(#OnTheFlyArcOn, WDAT1) DELAY = 0 DO ArcMainNG(#ArcOnMoveStd, WDAT1, WP3) PRIO = -1
  ArcMainNG(#ArcOnBeforeMoveStd, WDAT1, WP3)
  LIN XP3
  ArcMainNG(#ArcOnAfterMoveStd, WDAT1, WP3)
;ENDFOLD
   $VEL.CP = 0.030
   LIN  {X -1.918, Y 8.829, Z 0.300, A 0.000, B 0.000, C 0.000} C_DIS

;FOLD ARCOFF WDAT2 LIN P4 CPDAT2 Tool[1]:cmttorch Base[1]:vrashatel ;%{PE}
  ;FOLD Parameters ;%{h}
    ;Params IlfProvider=kukaroboter.arctech.arcofflin; Kuka.IsGlobalPoint=False; Kuka.PointName=P4; Kuka.BlendingEnabled=False; Kuka.MoveDataName=CPDAT2; Kuka.VelocityPath=0.01; Kuka.CurrentCDSetIndex=0; Kuka.MovementParameterFieldEnabled=True; ArcTech.WdatVarName=WDAT2; ArcTech.Basic=3.4.3.1264
  ;ENDFOLD
  $BWDSTART = FALSE
  LDAT_ACT = LCPDAT2
  FDAT_ACT = FP4
  BAS(#CP_PARAMS, gArcBasVelDefinition)
  SET_CD_PARAMS (0)
  TRIGGER WHEN PATH = ArcGetPath(#ArcOffBefore, WDAT2) DELAY = 0 DO ArcMainNG(#ArcOffBeforeOffStd, WDAT2, WP4) PRIO = -1
  TRIGGER WHEN PATH = ArcGetPath(#OnTheFlyArcOff, WDAT2) DELAY = 0 DO ArcMainNG(#ArcOffMoveStd, WDAT2, WP4) PRIO = -1
  ArcMainNG(#ArcOffBeforeMoveStd, WDAT2, WP4)
  LIN XP4
  ArcMainNG(#ArcOffAfterMoveStd, WDAT2, WP4)
;ENDFOLD
   $VEL.CP = 0.030
   LIN  {X -1.352, Y 8.829, Z 0.300, A 0.000, B 0.000, C 0.000} C_DIS

;FOLD ARCON WDAT1 LIN P3 Vel=0.5 m/s CPDAT1 Tool[1]:cmttorch Base[1]:vrashatel ;%{PE}
  ;FOLD Parameters ;%{h}
    ;Params IlfProvider=kukaroboter.arctech.arconlin; Kuka.IsGlobalPoint=False; Kuka.PointName=P3; Kuka.BlendingEnabled=False; Kuka.MoveDataName=CPDAT1; Kuka.VelocityPath=0.5; Kuka.CurrentCDSetIndex=0; Kuka.MovementParameterFieldEnabled=True; ArcTech.WdatVarName=WDAT1; ArcTech.Basic=3.4.3.1264
  ;ENDFOLD
  $BWDSTART = FALSE
  LDAT_ACT = LCPDAT1
  FDAT_ACT = FP3
  BAS(#CP_PARAMS, 0.5)
  SET_CD_PARAMS (0)
  TRIGGER WHEN DISTANCE = 1 DELAY = ArcGetDelay(#PreDefinition, WDAT1) DO ArcMainNG(#PreDefinition, WDAT1, WP3) PRIO = -1
  TRIGGER WHEN PATH = ArcGetPath(#OnTheFlyArcOn, WDAT1) DELAY = ArcGetDelay(#GasPreflow, WDAT1) DO ArcMainNG(#GasPreflow, WDAT1, WP3) PRIO = -1
  TRIGGER WHEN PATH = ArcGetPath(#OnTheFlyArcOn, WDAT1) DELAY = 0 DO ArcMainNG(#ArcOnMoveStd, WDAT1, WP3) PRIO = -1
  ArcMainNG(#ArcOnBeforeMoveStd, WDAT1, WP3)
  LIN XP3
  ArcMainNG(#ArcOnAfterMoveStd, WDAT1, WP3)
;ENDFOLD
   $VEL.CP = 0.030
   LIN  {X -8.829, Y 1.352, Z 0.300, A 0.000, B 0.000, C 0.000} C_DIS

;FOLD ARCOFF WDAT2 LIN P4 CPDAT2 Tool[1]:cmttorch Base[1]:vrashatel ;%{PE}
  ;FOLD Parameters ;%{h}
    ;Params IlfProvider=kukaroboter.arctech.arcofflin; Kuka.IsGlobalPoint=False; Kuka.PointName=P4; Kuka.BlendingEnabled=False; Kuka.MoveDataName=CPDAT2; Kuka.VelocityPath=0.01; Kuka.CurrentCDSetIndex=0; Kuka.MovementParameterFieldEnabled=True; ArcTech.WdatVarName=WDAT2; ArcTech.Basic=3.4.3.1264
  ;ENDFOLD
  $BWDSTART = FALSE
  LDAT_ACT = LCPDAT2
  FDAT_ACT = FP4
  BAS(#CP_PARAMS, gArcBasVelDefinition)
  SET_CD_PARAMS (0)
  TRIGGER WHEN PATH = ArcGetPath(#ArcOffBefore, WDAT2) DELAY = 0 DO ArcMainNG(#ArcOffBeforeOffStd, WDAT2, WP4) PRIO = -1
  TRIGGER WHEN PATH = ArcGetPath(#OnTheFlyArcOff, WDAT2) DELAY = 0 DO ArcMainNG(#ArcOffMoveStd, WDAT2, WP4) PRIO = -1
  ArcMainNG(#ArcOffBeforeMoveStd, WDAT2, WP4)
  LIN XP4
  ArcMainNG(#ArcOffAfterMoveStd, WDAT2, WP4)
;ENDFOLD
   $VEL.CP = 0.030
   LIN  {X -8.829, Y 0.787, Z 0.300, A 0.000, B 0.000, C 0.000} C_DIS

;FOLD ARCON WDAT1 LIN P3 Vel=0.5 m/s CPDAT1 Tool[1]:cmttorch Base[1]:vrashatel ;%{PE}
  ;FOLD Parameters ;%{h}
    ;Params IlfProvider=kukaroboter.arctech.arconlin; Kuka.IsGlobalPoint=False; Kuka.PointName=P3; Kuka.BlendingEnabled=False; Kuka.MoveDataName=CPDAT1; Kuka.VelocityPath=0.5; Kuka.CurrentCDSetIndex=0; Kuka.MovementParameterFieldEnabled=True; ArcTech.WdatVarName=WDAT1; ArcTech.Basic=3.4.3.1264
  ;ENDFOLD
  $BWDSTART = FALSE
  LDAT_ACT = LCPDAT1
  FDAT_ACT = FP3
  BAS(#CP_PARAMS, 0.5)
  SET_CD_PARAMS (0)
  TRIGGER WHEN DISTANCE = 1 DELAY = ArcGetDelay(#PreDefinition, WDAT1) DO ArcMainNG(#PreDefinition, WDAT1, WP3) PRIO = -1
  TRIGGER WHEN PATH = ArcGetPath(#OnTheFlyArcOn, WDAT1) DELAY = ArcGetDelay(#GasPreflow, WDAT1) DO ArcMainNG(#GasPreflow, WDAT1, WP3) PRIO = -1
  TRIGGER WHEN PATH = ArcGetPath(#OnTheFlyArcOn, WDAT1) DELAY = 0 DO ArcMainNG(#ArcOnMoveStd, WDAT1, WP3) PRIO = -1
  ArcMainNG(#ArcOnBeforeMoveStd, WDAT1, WP3)
  LIN XP3
  ArcMainNG(#ArcOnAfterMoveStd, WDAT1, WP3)
;ENDFOLD
   $VEL.CP = 0.030
   LIN  {X -0.787, Y 8.829, Z 0.300, A 0.000, B 0.000, C 0.000} C_DIS

;FOLD ARCOFF WDAT2 LIN P4 CPDAT2 Tool[1]:cmttorch Base[1]:vrashatel ;%{PE}
  ;FOLD Parameters ;%{h}
    ;Params IlfProvider=kukaroboter.arctech.arcofflin; Kuka.IsGlobalPoint=False; Kuka.PointName=P4; Kuka.BlendingEnabled=False; Kuka.MoveDataName=CPDAT2; Kuka.VelocityPath=0.01; Kuka.CurrentCDSetIndex=0; Kuka.MovementParameterFieldEnabled=True; ArcTech.WdatVarName=WDAT2; ArcTech.Basic=3.4.3.1264
  ;ENDFOLD
  $BWDSTART = FALSE
  LDAT_ACT = LCPDAT2
  FDAT_ACT = FP4
  BAS(#CP_PARAMS, gArcBasVelDefinition)
  SET_CD_PARAMS (0)
  TRIGGER WHEN PATH = ArcGetPath(#ArcOffBefore, WDAT2) DELAY = 0 DO ArcMainNG(#ArcOffBeforeOffStd, WDAT2, WP4) PRIO = -1
  TRIGGER WHEN PATH = ArcGetPath(#OnTheFlyArcOff, WDAT2) DELAY = 0 DO ArcMainNG(#ArcOffMoveStd, WDAT2, WP4) PRIO = -1
  ArcMainNG(#ArcOffBeforeMoveStd, WDAT2, WP4)
  LIN XP4
  ArcMainNG(#ArcOffAfterMoveStd, WDAT2, WP4)
;ENDFOLD
   $VEL.CP = 0.030
   LIN  {X -0.221, Y 8.829, Z 0.300, A 0.000, B 0.000, C 0.000} C_DIS

;FOLD ARCON WDAT1 LIN P3 Vel=0.5 m/s CPDAT1 Tool[1]:cmttorch Base[1]:vrashatel ;%{PE}
  ;FOLD Parameters ;%{h}
    ;Params IlfProvider=kukaroboter.arctech.arconlin; Kuka.IsGlobalPoint=False; Kuka.PointName=P3; Kuka.BlendingEnabled=False; Kuka.MoveDataName=CPDAT1; Kuka.VelocityPath=0.5; Kuka.CurrentCDSetIndex=0; Kuka.MovementParameterFieldEnabled=True; ArcTech.WdatVarName=WDAT1; ArcTech.Basic=3.4.3.1264
  ;ENDFOLD
  $BWDSTART = FALSE
  LDAT_ACT = LCPDAT1
  FDAT_ACT = FP3
  BAS(#CP_PARAMS, 0.5)
  SET_CD_PARAMS (0)
  TRIGGER WHEN DISTANCE = 1 DELAY = ArcGetDelay(#PreDefinition, WDAT1) DO ArcMainNG(#PreDefinition, WDAT1, WP3) PRIO = -1
  TRIGGER WHEN PATH = ArcGetPath(#OnTheFlyArcOn, WDAT1) DELAY = ArcGetDelay(#GasPreflow, WDAT1) DO ArcMainNG(#GasPreflow, WDAT1, WP3) PRIO = -1
  TRIGGER WHEN PATH = ArcGetPath(#OnTheFlyArcOn, WDAT1) DELAY = 0 DO ArcMainNG(#ArcOnMoveStd, WDAT1, WP3) PRIO = -1
  ArcMainNG(#ArcOnBeforeMoveStd, WDAT1, WP3)
  LIN XP3
  ArcMainNG(#ArcOnAfterMoveStd, WDAT1, WP3)
;ENDFOLD
   $VEL.CP = 0.030
   LIN  {X -8.829, Y 0.221, Z 0.300, A 0.000, B 0.000, C 0.000} C_DIS

;FOLD ARCOFF WDAT2 LIN P4 CPDAT2 Tool[1]:cmttorch Base[1]:vrashatel ;%{PE}
  ;FOLD Parameters ;%{h}
    ;Params IlfProvider=kukaroboter.arctech.arcofflin; Kuka.IsGlobalPoint=False; Kuka.PointName=P4; Kuka.BlendingEnabled=False; Kuka.MoveDataName=CPDAT2; Kuka.VelocityPath=0.01; Kuka.CurrentCDSetIndex=0; Kuka.MovementParameterFieldEnabled=True; ArcTech.WdatVarName=WDAT2; ArcTech.Basic=3.4.3.1264
  ;ENDFOLD
  $BWDSTART = FALSE
  LDAT_ACT = LCPDAT2
  FDAT_ACT = FP4
  BAS(#CP_PARAMS, gArcBasVelDefinition)
  SET_CD_PARAMS (0)
  TRIGGER WHEN PATH = ArcGetPath(#ArcOffBefore, WDAT2) DELAY = 0 DO ArcMainNG(#ArcOffBeforeOffStd, WDAT2, WP4) PRIO = -1
  TRIGGER WHEN PATH = ArcGetPath(#OnTheFlyArcOff, WDAT2) DELAY = 0 DO ArcMainNG(#ArcOffMoveStd, WDAT2, WP4) PRIO = -1
  ArcMainNG(#ArcOffBeforeMoveStd, WDAT2, WP4)
  LIN XP4
  ArcMainNG(#ArcOffAfterMoveStd, WDAT2, WP4)
;ENDFOLD
   $VEL.CP = 0.030
   LIN  {X -8.829, Y -0.344, Z 0.300, A 0.000, B 0.000, C 0.000} C_DIS

;FOLD ARCON WDAT1 LIN P3 Vel=0.5 m/s CPDAT1 Tool[1]:cmttorch Base[1]:vrashatel ;%{PE}
  ;FOLD Parameters ;%{h}
    ;Params IlfProvider=kukaroboter.arctech.arconlin; Kuka.IsGlobalPoint=False; Kuka.PointName=P3; Kuka.BlendingEnabled=False; Kuka.MoveDataName=CPDAT1; Kuka.VelocityPath=0.5; Kuka.CurrentCDSetIndex=0; Kuka.MovementParameterFieldEnabled=True; ArcTech.WdatVarName=WDAT1; ArcTech.Basic=3.4.3.1264
  ;ENDFOLD
  $BWDSTART = FALSE
  LDAT_ACT = LCPDAT1
  FDAT_ACT = FP3
  BAS(#CP_PARAMS, 0.5)
  SET_CD_PARAMS (0)
  TRIGGER WHEN DISTANCE = 1 DELAY = ArcGetDelay(#PreDefinition, WDAT1) DO ArcMainNG(#PreDefinition, WDAT1, WP3) PRIO = -1
  TRIGGER WHEN PATH = ArcGetPath(#OnTheFlyArcOn, WDAT1) DELAY = ArcGetDelay(#GasPreflow, WDAT1) DO ArcMainNG(#GasPreflow, WDAT1, WP3) PRIO = -1
  TRIGGER WHEN PATH = ArcGetPath(#OnTheFlyArcOn, WDAT1) DELAY = 0 DO ArcMainNG(#ArcOnMoveStd, WDAT1, WP3) PRIO = -1
  ArcMainNG(#ArcOnBeforeMoveStd, WDAT1, WP3)
  LIN XP3
  ArcMainNG(#ArcOnAfterMoveStd, WDAT1, WP3)
;ENDFOLD
   $VEL.CP = 0.030
   LIN  {X 0.344, Y 8.829, Z 0.300, A 0.000, B 0.000, C 0.000} C_DIS

;FOLD ARCOFF WDAT2 LIN P4 CPDAT2 Tool[1]:cmttorch Base[1]:vrashatel ;%{PE}
  ;FOLD Parameters ;%{h}
    ;Params IlfProvider=kukaroboter.arctech.arcofflin; Kuka.IsGlobalPoint=False; Kuka.PointName=P4; Kuka.BlendingEnabled=False; Kuka.MoveDataName=CPDAT2; Kuka.VelocityPath=0.01; Kuka.CurrentCDSetIndex=0; Kuka.MovementParameterFieldEnabled=True; ArcTech.WdatVarName=WDAT2; ArcTech.Basic=3.4.3.1264
  ;ENDFOLD
  $BWDSTART = FALSE
  LDAT_ACT = LCPDAT2
  FDAT_ACT = FP4
  BAS(#CP_PARAMS, gArcBasVelDefinition)
  SET_CD_PARAMS (0)
  TRIGGER WHEN PATH = ArcGetPath(#ArcOffBefore, WDAT2) DELAY = 0 DO ArcMainNG(#ArcOffBeforeOffStd, WDAT2, WP4) PRIO = -1
  TRIGGER WHEN PATH = ArcGetPath(#OnTheFlyArcOff, WDAT2) DELAY = 0 DO ArcMainNG(#ArcOffMoveStd, WDAT2, WP4) PRIO = -1
  ArcMainNG(#ArcOffBeforeMoveStd, WDAT2, WP4)
  LIN XP4
  ArcMainNG(#ArcOffAfterMoveStd, WDAT2, WP4)
;ENDFOLD
   $VEL.CP = 0.030
   LIN  {X 0.910, Y 8.829, Z 0.300, A 0.000, B 0.000, C 0.000} C_DIS

;FOLD ARCON WDAT1 LIN P3 Vel=0.5 m/s CPDAT1 Tool[1]:cmttorch Base[1]:vrashatel ;%{PE}
  ;FOLD Parameters ;%{h}
    ;Params IlfProvider=kukaroboter.arctech.arconlin; Kuka.IsGlobalPoint=False; Kuka.PointName=P3; Kuka.BlendingEnabled=False; Kuka.MoveDataName=CPDAT1; Kuka.VelocityPath=0.5; Kuka.CurrentCDSetIndex=0; Kuka.MovementParameterFieldEnabled=True; ArcTech.WdatVarName=WDAT1; ArcTech.Basic=3.4.3.1264
  ;ENDFOLD
  $BWDSTART = FALSE
  LDAT_ACT = LCPDAT1
  FDAT_ACT = FP3
  BAS(#CP_PARAMS, 0.5)
  SET_CD_PARAMS (0)
  TRIGGER WHEN DISTANCE = 1 DELAY = ArcGetDelay(#PreDefinition, WDAT1) DO ArcMainNG(#PreDefinition, WDAT1, WP3) PRIO = -1
  TRIGGER WHEN PATH = ArcGetPath(#OnTheFlyArcOn, WDAT1) DELAY = ArcGetDelay(#GasPreflow, WDAT1) DO ArcMainNG(#GasPreflow, WDAT1, WP3) PRIO = -1
  TRIGGER WHEN PATH = ArcGetPath(#OnTheFlyArcOn, WDAT1) DELAY = 0 DO ArcMainNG(#ArcOnMoveStd, WDAT1, WP3) PRIO = -1
  ArcMainNG(#ArcOnBeforeMoveStd, WDAT1, WP3)
  LIN XP3
  ArcMainNG(#ArcOnAfterMoveStd, WDAT1, WP3)
;ENDFOLD
   $VEL.CP = 0.030
   LIN  {X -8.829, Y -0.910, Z 0.300, A 0.000, B 0.000, C 0.000} C_DIS

;FOLD ARCOFF WDAT2 LIN P4 CPDAT2 Tool[1]:cmttorch Base[1]:vrashatel ;%{PE}
  ;FOLD Parameters ;%{h}
    ;Params IlfProvider=kukaroboter.arctech.arcofflin; Kuka.IsGlobalPoint=False; Kuka.PointName=P4; Kuka.BlendingEnabled=False; Kuka.MoveDataName=CPDAT2; Kuka.VelocityPath=0.01; Kuka.CurrentCDSetIndex=0; Kuka.MovementParameterFieldEnabled=True; ArcTech.WdatVarName=WDAT2; ArcTech.Basic=3.4.3.1264
  ;ENDFOLD
  $BWDSTART = FALSE
  LDAT_ACT = LCPDAT2
  FDAT_ACT = FP4
  BAS(#CP_PARAMS, gArcBasVelDefinition)
  SET_CD_PARAMS (0)
  TRIGGER WHEN PATH = ArcGetPath(#ArcOffBefore, WDAT2) DELAY = 0 DO ArcMainNG(#ArcOffBeforeOffStd, WDAT2, WP4) PRIO = -1
  TRIGGER WHEN PATH = ArcGetPath(#OnTheFlyArcOff, WDAT2) DELAY = 0 DO ArcMainNG(#ArcOffMoveStd, WDAT2, WP4) PRIO = -1
  ArcMainNG(#ArcOffBeforeMoveStd, WDAT2, WP4)
  LIN XP4
  ArcMainNG(#ArcOffAfterMoveStd, WDAT2, WP4)
;ENDFOLD
   $VEL.CP = 0.030
   LIN  {X -8.829, Y -1.475, Z 0.300, A 0.000, B 0.000, C 0.000} C_DIS

;FOLD ARCON WDAT1 LIN P3 Vel=0.5 m/s CPDAT1 Tool[1]:cmttorch Base[1]:vrashatel ;%{PE}
  ;FOLD Parameters ;%{h}
    ;Params IlfProvider=kukaroboter.arctech.arconlin; Kuka.IsGlobalPoint=False; Kuka.PointName=P3; Kuka.BlendingEnabled=False; Kuka.MoveDataName=CPDAT1; Kuka.VelocityPath=0.5; Kuka.CurrentCDSetIndex=0; Kuka.MovementParameterFieldEnabled=True; ArcTech.WdatVarName=WDAT1; ArcTech.Basic=3.4.3.1264
  ;ENDFOLD
  $BWDSTART = FALSE
  LDAT_ACT = LCPDAT1
  FDAT_ACT = FP3
  BAS(#CP_PARAMS, 0.5)
  SET_CD_PARAMS (0)
  TRIGGER WHEN DISTANCE = 1 DELAY = ArcGetDelay(#PreDefinition, WDAT1) DO ArcMainNG(#PreDefinition, WDAT1, WP3) PRIO = -1
  TRIGGER WHEN PATH = ArcGetPath(#OnTheFlyArcOn, WDAT1) DELAY = ArcGetDelay(#GasPreflow, WDAT1) DO ArcMainNG(#GasPreflow, WDAT1, WP3) PRIO = -1
  TRIGGER WHEN PATH = ArcGetPath(#OnTheFlyArcOn, WDAT1) DELAY = 0 DO ArcMainNG(#ArcOnMoveStd, WDAT1, WP3) PRIO = -1
  ArcMainNG(#ArcOnBeforeMoveStd, WDAT1, WP3)
  LIN XP3
  ArcMainNG(#ArcOnAfterMoveStd, WDAT1, WP3)
;ENDFOLD
   $VEL.CP = 0.030
   LIN  {X 1.475, Y 8.829, Z 0.300, A 0.000, B 0.000, C 0.000} C_DIS

;FOLD ARCOFF WDAT2 LIN P4 CPDAT2 Tool[1]:cmttorch Base[1]:vrashatel ;%{PE}
  ;FOLD Parameters ;%{h}
    ;Params IlfProvider=kukaroboter.arctech.arcofflin; Kuka.IsGlobalPoint=False; Kuka.PointName=P4; Kuka.BlendingEnabled=False; Kuka.MoveDataName=CPDAT2; Kuka.VelocityPath=0.01; Kuka.CurrentCDSetIndex=0; Kuka.MovementParameterFieldEnabled=True; ArcTech.WdatVarName=WDAT2; ArcTech.Basic=3.4.3.1264
  ;ENDFOLD
  $BWDSTART = FALSE
  LDAT_ACT = LCPDAT2
  FDAT_ACT = FP4
  BAS(#CP_PARAMS, gArcBasVelDefinition)
  SET_CD_PARAMS (0)
  TRIGGER WHEN PATH = ArcGetPath(#ArcOffBefore, WDAT2) DELAY = 0 DO ArcMainNG(#ArcOffBeforeOffStd, WDAT2, WP4) PRIO = -1
  TRIGGER WHEN PATH = ArcGetPath(#OnTheFlyArcOff, WDAT2) DELAY = 0 DO ArcMainNG(#ArcOffMoveStd, WDAT2, WP4) PRIO = -1
  ArcMainNG(#ArcOffBeforeMoveStd, WDAT2, WP4)
  LIN XP4
  ArcMainNG(#ArcOffAfterMoveStd, WDAT2, WP4)
;ENDFOLD
   $VEL.CP = 0.030
   LIN  {X 2.041, Y 8.829, Z 0.300, A 0.000, B 0.000, C 0.000} C_DIS

;FOLD ARCON WDAT1 LIN P3 Vel=0.5 m/s CPDAT1 Tool[1]:cmttorch Base[1]:vrashatel ;%{PE}
  ;FOLD Parameters ;%{h}
    ;Params IlfProvider=kukaroboter.arctech.arconlin; Kuka.IsGlobalPoint=False; Kuka.PointName=P3; Kuka.BlendingEnabled=False; Kuka.MoveDataName=CPDAT1; Kuka.VelocityPath=0.5; Kuka.CurrentCDSetIndex=0; Kuka.MovementParameterFieldEnabled=True; ArcTech.WdatVarName=WDAT1; ArcTech.Basic=3.4.3.1264
  ;ENDFOLD
  $BWDSTART = FALSE
  LDAT_ACT = LCPDAT1
  FDAT_ACT = FP3
  BAS(#CP_PARAMS, 0.5)
  SET_CD_PARAMS (0)
  TRIGGER WHEN DISTANCE = 1 DELAY = ArcGetDelay(#PreDefinition, WDAT1) DO ArcMainNG(#PreDefinition, WDAT1, WP3) PRIO = -1
  TRIGGER WHEN PATH = ArcGetPath(#OnTheFlyArcOn, WDAT1) DELAY = ArcGetDelay(#GasPreflow, WDAT1) DO ArcMainNG(#GasPreflow, WDAT1, WP3) PRIO = -1
  TRIGGER WHEN PATH = ArcGetPath(#OnTheFlyArcOn, WDAT1) DELAY = 0 DO ArcMainNG(#ArcOnMoveStd, WDAT1, WP3) PRIO = -1
  ArcMainNG(#ArcOnBeforeMoveStd, WDAT1, WP3)
  LIN XP3
  ArcMainNG(#ArcOnAfterMoveStd, WDAT1, WP3)
;ENDFOLD
   $VEL.CP = 0.030
   LIN  {X -8.829, Y -2.041, Z 0.300, A 0.000, B 0.000, C 0.000} C_DIS

;FOLD ARCOFF WDAT2 LIN P4 CPDAT2 Tool[1]:cmttorch Base[1]:vrashatel ;%{PE}
  ;FOLD Parameters ;%{h}
    ;Params IlfProvider=kukaroboter.arctech.arcofflin; Kuka.IsGlobalPoint=False; Kuka.PointName=P4; Kuka.BlendingEnabled=False; Kuka.MoveDataName=CPDAT2; Kuka.VelocityPath=0.01; Kuka.CurrentCDSetIndex=0; Kuka.MovementParameterFieldEnabled=True; ArcTech.WdatVarName=WDAT2; ArcTech.Basic=3.4.3.1264
  ;ENDFOLD
  $BWDSTART = FALSE
  LDAT_ACT = LCPDAT2
  FDAT_ACT = FP4
  BAS(#CP_PARAMS, gArcBasVelDefinition)
  SET_CD_PARAMS (0)
  TRIGGER WHEN PATH = ArcGetPath(#ArcOffBefore, WDAT2) DELAY = 0 DO ArcMainNG(#ArcOffBeforeOffStd, WDAT2, WP4) PRIO = -1
  TRIGGER WHEN PATH = ArcGetPath(#OnTheFlyArcOff, WDAT2) DELAY = 0 DO ArcMainNG(#ArcOffMoveStd, WDAT2, WP4) PRIO = -1
  ArcMainNG(#ArcOffBeforeMoveStd, WDAT2, WP4)
  LIN XP4
  ArcMainNG(#ArcOffAfterMoveStd, WDAT2, WP4)
;ENDFOLD
   $VEL.CP = 0.030
   LIN  {X -8.829, Y -2.607, Z 0.300, A 0.000, B 0.000, C 0.000} C_DIS

;FOLD ARCON WDAT1 LIN P3 Vel=0.5 m/s CPDAT1 Tool[1]:cmttorch Base[1]:vrashatel ;%{PE}
  ;FOLD Parameters ;%{h}
    ;Params IlfProvider=kukaroboter.arctech.arconlin; Kuka.IsGlobalPoint=False; Kuka.PointName=P3; Kuka.BlendingEnabled=False; Kuka.MoveDataName=CPDAT1; Kuka.VelocityPath=0.5; Kuka.CurrentCDSetIndex=0; Kuka.MovementParameterFieldEnabled=True; ArcTech.WdatVarName=WDAT1; ArcTech.Basic=3.4.3.1264
  ;ENDFOLD
  $BWDSTART = FALSE
  LDAT_ACT = LCPDAT1
  FDAT_ACT = FP3
  BAS(#CP_PARAMS, 0.5)
  SET_CD_PARAMS (0)
  TRIGGER WHEN DISTANCE = 1 DELAY = ArcGetDelay(#PreDefinition, WDAT1) DO ArcMainNG(#PreDefinition, WDAT1, WP3) PRIO = -1
  TRIGGER WHEN PATH = ArcGetPath(#OnTheFlyArcOn, WDAT1) DELAY = ArcGetDelay(#GasPreflow, WDAT1) DO ArcMainNG(#GasPreflow, WDAT1, WP3) PRIO = -1
  TRIGGER WHEN PATH = ArcGetPath(#OnTheFlyArcOn, WDAT1) DELAY = 0 DO ArcMainNG(#ArcOnMoveStd, WDAT1, WP3) PRIO = -1
  ArcMainNG(#ArcOnBeforeMoveStd, WDAT1, WP3)
  LIN XP3
  ArcMainNG(#ArcOnAfterMoveStd, WDAT1, WP3)
;ENDFOLD
   $VEL.CP = 0.030
   LIN  {X 2.607, Y 8.829, Z 0.300, A 0.000, B 0.000, C 0.000} C_DIS

;FOLD ARCOFF WDAT2 LIN P4 CPDAT2 Tool[1]:cmttorch Base[1]:vrashatel ;%{PE}
  ;FOLD Parameters ;%{h}
    ;Params IlfProvider=kukaroboter.arctech.arcofflin; Kuka.IsGlobalPoint=False; Kuka.PointName=P4; Kuka.BlendingEnabled=False; Kuka.MoveDataName=CPDAT2; Kuka.VelocityPath=0.01; Kuka.CurrentCDSetIndex=0; Kuka.MovementParameterFieldEnabled=True; ArcTech.WdatVarName=WDAT2; ArcTech.Basic=3.4.3.1264
  ;ENDFOLD
  $BWDSTART = FALSE
  LDAT_ACT = LCPDAT2
  FDAT_ACT = FP4
  BAS(#CP_PARAMS, gArcBasVelDefinition)
  SET_CD_PARAMS (0)
  TRIGGER WHEN PATH = ArcGetPath(#ArcOffBefore, WDAT2) DELAY = 0 DO ArcMainNG(#ArcOffBeforeOffStd, WDAT2, WP4) PRIO = -1
  TRIGGER WHEN PATH = ArcGetPath(#OnTheFlyArcOff, WDAT2) DELAY = 0 DO ArcMainNG(#ArcOffMoveStd, WDAT2, WP4) PRIO = -1
  ArcMainNG(#ArcOffBeforeMoveStd, WDAT2, WP4)
  LIN XP4
  ArcMainNG(#ArcOffAfterMoveStd, WDAT2, WP4)
;ENDFOLD
   $VEL.CP = 0.030
   LIN  {X 3.172, Y 8.829, Z 0.300, A 0.000, B 0.000, C 0.000} C_DIS

;FOLD ARCON WDAT1 LIN P3 Vel=0.5 m/s CPDAT1 Tool[1]:cmttorch Base[1]:vrashatel ;%{PE}
  ;FOLD Parameters ;%{h}
    ;Params IlfProvider=kukaroboter.arctech.arconlin; Kuka.IsGlobalPoint=False; Kuka.PointName=P3; Kuka.BlendingEnabled=False; Kuka.MoveDataName=CPDAT1; Kuka.VelocityPath=0.5; Kuka.CurrentCDSetIndex=0; Kuka.MovementParameterFieldEnabled=True; ArcTech.WdatVarName=WDAT1; ArcTech.Basic=3.4.3.1264
  ;ENDFOLD
  $BWDSTART = FALSE
  LDAT_ACT = LCPDAT1
  FDAT_ACT = FP3
  BAS(#CP_PARAMS, 0.5)
  SET_CD_PARAMS (0)
  TRIGGER WHEN DISTANCE = 1 DELAY = ArcGetDelay(#PreDefinition, WDAT1) DO ArcMainNG(#PreDefinition, WDAT1, WP3) PRIO = -1
  TRIGGER WHEN PATH = ArcGetPath(#OnTheFlyArcOn, WDAT1) DELAY = ArcGetDelay(#GasPreflow, WDAT1) DO ArcMainNG(#GasPreflow, WDAT1, WP3) PRIO = -1
  TRIGGER WHEN PATH = ArcGetPath(#OnTheFlyArcOn, WDAT1) DELAY = 0 DO ArcMainNG(#ArcOnMoveStd, WDAT1, WP3) PRIO = -1
  ArcMainNG(#ArcOnBeforeMoveStd, WDAT1, WP3)
  LIN XP3
  ArcMainNG(#ArcOnAfterMoveStd, WDAT1, WP3)
;ENDFOLD
   $VEL.CP = 0.030
   LIN  {X -8.829, Y -3.172, Z 0.300, A 0.000, B 0.000, C 0.000} C_DIS

;FOLD ARCOFF WDAT2 LIN P4 CPDAT2 Tool[1]:cmttorch Base[1]:vrashatel ;%{PE}
  ;FOLD Parameters ;%{h}
    ;Params IlfProvider=kukaroboter.arctech.arcofflin; Kuka.IsGlobalPoint=False; Kuka.PointName=P4; Kuka.BlendingEnabled=False; Kuka.MoveDataName=CPDAT2; Kuka.VelocityPath=0.01; Kuka.CurrentCDSetIndex=0; Kuka.MovementParameterFieldEnabled=True; ArcTech.WdatVarName=WDAT2; ArcTech.Basic=3.4.3.1264
  ;ENDFOLD
  $BWDSTART = FALSE
  LDAT_ACT = LCPDAT2
  FDAT_ACT = FP4
  BAS(#CP_PARAMS, gArcBasVelDefinition)
  SET_CD_PARAMS (0)
  TRIGGER WHEN PATH = ArcGetPath(#ArcOffBefore, WDAT2) DELAY = 0 DO ArcMainNG(#ArcOffBeforeOffStd, WDAT2, WP4) PRIO = -1
  TRIGGER WHEN PATH = ArcGetPath(#OnTheFlyArcOff, WDAT2) DELAY = 0 DO ArcMainNG(#ArcOffMoveStd, WDAT2, WP4) PRIO = -1
  ArcMainNG(#ArcOffBeforeMoveStd, WDAT2, WP4)
  LIN XP4
  ArcMainNG(#ArcOffAfterMoveStd, WDAT2, WP4)
;ENDFOLD
   $VEL.CP = 0.030
   LIN  {X -8.829, Y -3.738, Z 0.300, A 0.000, B 0.000, C 0.000} C_DIS

;FOLD ARCON WDAT1 LIN P3 Vel=0.5 m/s CPDAT1 Tool[1]:cmttorch Base[1]:vrashatel ;%{PE}
  ;FOLD Parameters ;%{h}
    ;Params IlfProvider=kukaroboter.arctech.arconlin; Kuka.IsGlobalPoint=False; Kuka.PointName=P3; Kuka.BlendingEnabled=False; Kuka.MoveDataName=CPDAT1; Kuka.VelocityPath=0.5; Kuka.CurrentCDSetIndex=0; Kuka.MovementParameterFieldEnabled=True; ArcTech.WdatVarName=WDAT1; ArcTech.Basic=3.4.3.1264
  ;ENDFOLD
  $BWDSTART = FALSE
  LDAT_ACT = LCPDAT1
  FDAT_ACT = FP3
  BAS(#CP_PARAMS, 0.5)
  SET_CD_PARAMS (0)
  TRIGGER WHEN DISTANCE = 1 DELAY = ArcGetDelay(#PreDefinition, WDAT1) DO ArcMainNG(#PreDefinition, WDAT1, WP3) PRIO = -1
  TRIGGER WHEN PATH = ArcGetPath(#OnTheFlyArcOn, WDAT1) DELAY = ArcGetDelay(#GasPreflow, WDAT1) DO ArcMainNG(#GasPreflow, WDAT1, WP3) PRIO = -1
  TRIGGER WHEN PATH = ArcGetPath(#OnTheFlyArcOn, WDAT1) DELAY = 0 DO ArcMainNG(#ArcOnMoveStd, WDAT1, WP3) PRIO = -1
  ArcMainNG(#ArcOnBeforeMoveStd, WDAT1, WP3)
  LIN XP3
  ArcMainNG(#ArcOnAfterMoveStd, WDAT1, WP3)
;ENDFOLD
   $VEL.CP = 0.030
   LIN  {X 3.738, Y 8.829, Z 0.300, A 0.000, B 0.000, C 0.000} C_DIS

;FOLD ARCOFF WDAT2 LIN P4 CPDAT2 Tool[1]:cmttorch Base[1]:vrashatel ;%{PE}
  ;FOLD Parameters ;%{h}
    ;Params IlfProvider=kukaroboter.arctech.arcofflin; Kuka.IsGlobalPoint=False; Kuka.PointName=P4; Kuka.BlendingEnabled=False; Kuka.MoveDataName=CPDAT2; Kuka.VelocityPath=0.01; Kuka.CurrentCDSetIndex=0; Kuka.MovementParameterFieldEnabled=True; ArcTech.WdatVarName=WDAT2; ArcTech.Basic=3.4.3.1264
  ;ENDFOLD
  $BWDSTART = FALSE
  LDAT_ACT = LCPDAT2
  FDAT_ACT = FP4
  BAS(#CP_PARAMS, gArcBasVelDefinition)
  SET_CD_PARAMS (0)
  TRIGGER WHEN PATH = ArcGetPath(#ArcOffBefore, WDAT2) DELAY = 0 DO ArcMainNG(#ArcOffBeforeOffStd, WDAT2, WP4) PRIO = -1
  TRIGGER WHEN PATH = ArcGetPath(#OnTheFlyArcOff, WDAT2) DELAY = 0 DO ArcMainNG(#ArcOffMoveStd, WDAT2, WP4) PRIO = -1
  ArcMainNG(#ArcOffBeforeMoveStd, WDAT2, WP4)
  LIN XP4
  ArcMainNG(#ArcOffAfterMoveStd, WDAT2, WP4)
;ENDFOLD
   $VEL.CP = 0.030
   LIN  {X 4.304, Y 8.829, Z 0.300, A 0.000, B 0.000, C 0.000} C_DIS

;FOLD ARCON WDAT1 LIN P3 Vel=0.5 m/s CPDAT1 Tool[1]:cmttorch Base[1]:vrashatel ;%{PE}
  ;FOLD Parameters ;%{h}
    ;Params IlfProvider=kukaroboter.arctech.arconlin; Kuka.IsGlobalPoint=False; Kuka.PointName=P3; Kuka.BlendingEnabled=False; Kuka.MoveDataName=CPDAT1; Kuka.VelocityPath=0.5; Kuka.CurrentCDSetIndex=0; Kuka.MovementParameterFieldEnabled=True; ArcTech.WdatVarName=WDAT1; ArcTech.Basic=3.4.3.1264
  ;ENDFOLD
  $BWDSTART = FALSE
  LDAT_ACT = LCPDAT1
  FDAT_ACT = FP3
  BAS(#CP_PARAMS, 0.5)
  SET_CD_PARAMS (0)
  TRIGGER WHEN DISTANCE = 1 DELAY = ArcGetDelay(#PreDefinition, WDAT1) DO ArcMainNG(#PreDefinition, WDAT1, WP3) PRIO = -1
  TRIGGER WHEN PATH = ArcGetPath(#OnTheFlyArcOn, WDAT1) DELAY = ArcGetDelay(#GasPreflow, WDAT1) DO ArcMainNG(#GasPreflow, WDAT1, WP3) PRIO = -1
  TRIGGER WHEN PATH = ArcGetPath(#OnTheFlyArcOn, WDAT1) DELAY = 0 DO ArcMainNG(#ArcOnMoveStd, WDAT1, WP3) PRIO = -1
  ArcMainNG(#ArcOnBeforeMoveStd, WDAT1, WP3)
  LIN XP3
  ArcMainNG(#ArcOnAfterMoveStd, WDAT1, WP3)
;ENDFOLD
   $VEL.CP = 0.030
   LIN  {X -8.829, Y -4.304, Z 0.300, A 0.000, B 0.000, C 0.000} C_DIS

;FOLD ARCOFF WDAT2 LIN P4 CPDAT2 Tool[1]:cmttorch Base[1]:vrashatel ;%{PE}
  ;FOLD Parameters ;%{h}
    ;Params IlfProvider=kukaroboter.arctech.arcofflin; Kuka.IsGlobalPoint=False; Kuka.PointName=P4; Kuka.BlendingEnabled=False; Kuka.MoveDataName=CPDAT2; Kuka.VelocityPath=0.01; Kuka.CurrentCDSetIndex=0; Kuka.MovementParameterFieldEnabled=True; ArcTech.WdatVarName=WDAT2; ArcTech.Basic=3.4.3.1264
  ;ENDFOLD
  $BWDSTART = FALSE
  LDAT_ACT = LCPDAT2
  FDAT_ACT = FP4
  BAS(#CP_PARAMS, gArcBasVelDefinition)
  SET_CD_PARAMS (0)
  TRIGGER WHEN PATH = ArcGetPath(#ArcOffBefore, WDAT2) DELAY = 0 DO ArcMainNG(#ArcOffBeforeOffStd, WDAT2, WP4) PRIO = -1
  TRIGGER WHEN PATH = ArcGetPath(#OnTheFlyArcOff, WDAT2) DELAY = 0 DO ArcMainNG(#ArcOffMoveStd, WDAT2, WP4) PRIO = -1
  ArcMainNG(#ArcOffBeforeMoveStd, WDAT2, WP4)
  LIN XP4
  ArcMainNG(#ArcOffAfterMoveStd, WDAT2, WP4)
;ENDFOLD
   $VEL.CP = 0.030
   LIN  {X -8.829, Y -4.869, Z 0.300, A 0.000, B 0.000, C 0.000} C_DIS

;FOLD ARCON WDAT1 LIN P3 Vel=0.5 m/s CPDAT1 Tool[1]:cmttorch Base[1]:vrashatel ;%{PE}
  ;FOLD Parameters ;%{h}
    ;Params IlfProvider=kukaroboter.arctech.arconlin; Kuka.IsGlobalPoint=False; Kuka.PointName=P3; Kuka.BlendingEnabled=False; Kuka.MoveDataName=CPDAT1; Kuka.VelocityPath=0.5; Kuka.CurrentCDSetIndex=0; Kuka.MovementParameterFieldEnabled=True; ArcTech.WdatVarName=WDAT1; ArcTech.Basic=3.4.3.1264
  ;ENDFOLD
  $BWDSTART = FALSE
  LDAT_ACT = LCPDAT1
  FDAT_ACT = FP3
  BAS(#CP_PARAMS, 0.5)
  SET_CD_PARAMS (0)
  TRIGGER WHEN DISTANCE = 1 DELAY = ArcGetDelay(#PreDefinition, WDAT1) DO ArcMainNG(#PreDefinition, WDAT1, WP3) PRIO = -1
  TRIGGER WHEN PATH = ArcGetPath(#OnTheFlyArcOn, WDAT1) DELAY = ArcGetDelay(#GasPreflow, WDAT1) DO ArcMainNG(#GasPreflow, WDAT1, WP3) PRIO = -1
  TRIGGER WHEN PATH = ArcGetPath(#OnTheFlyArcOn, WDAT1) DELAY = 0 DO ArcMainNG(#ArcOnMoveStd, WDAT1, WP3) PRIO = -1
  ArcMainNG(#ArcOnBeforeMoveStd, WDAT1, WP3)
  LIN XP3
  ArcMainNG(#ArcOnAfterMoveStd, WDAT1, WP3)
;ENDFOLD
   $VEL.CP = 0.030
   LIN  {X 4.869, Y 8.829, Z 0.300, A 0.000, B 0.000, C 0.000} C_DIS

